ATQ.Height := 150;
ATQ.Length := 800; //1200;
ATQ.Weight := 1500;
ATQ.Width := 800;
ATQ.LabelPresent := 1;
ATQ.Label := CONCAT('TESTLABEL_',NewID);

fbITC_ManagerEmulation.M_AddData(
	meChannelSrc := 0,
	mMsgType     := E_ITC_MsgTypeConv.E_ADD_TU_REQUEST,
	mpData		 := ADR(ATQ),
    mLen 		 := SIZEOF(ATQ));

END_FUNCTION

// ---- 20_Product/20_ProBox/30_Toolbox/11_Emu/F_RemovePhysicalTU.TcPOU
FUNCTION F_RemovePhysicalTU : BOOL
(**************************************************************************************
 * 	Application		:	BoxControl Framework
 *	Revision		:	$Revision: 353897 $
 *	Revision date	:	$Date: 2015-08-24 22:28:50 +0200 (Mo, 24 Aug 2015) $
 *	Last changed by	:	$Author: d7mangc $
 *	URL				:	$URL: http://almscdc.swisslog.com/repo/SWPD/Development/BoxControlFramework/20_Release/trunk/01_Software/BoxControlFramework/BoxControlFramework/JumpStart/11_Library/10_Application/12_ElementFunctions/10_Functions/F_GetFunctionData.TcPOU $
 *
 *	Purpose			:	Removes physical (emulation) TU data
 *
 * ------------------------------------------------------------------------------------
 *	Copyright Swisslog [IP AG], Switzerland. All rights reserved.
 * 
 * ------------------------------------------------------------------------------------
 *	
 * 	Revision History: 
 *
 * 	VERSION			DATE			INITIALS			DESCRIPTION
 *	0.1				01.01.2001		swl					Example
 *
 **************************************************************************************)
VAR_INPUT
	eFunctionNumber : E_FunctionNumber;
	ZoneNumber		: INT;
END_VAR
VAR
	Name			: STRING;
	RTQ				: ST_ITC_RTQ;
	TransportData	: ST_TransportControlData;
END_VAR

TransportData := F_GetTransportControlData(eFunctionNumber, ZoneNumber);

IF TransportData.SensorOccupied THEN
	Name := F_GetFunctionName(eFunctionNumber:= eFunctionNumber, ZoneNumber:= ZoneNumber);
	RTQ.Position := F_ReduceToAlphaNumeric(InputString := Name);
	
	fbITC_ManagerEmulation.M_AddData(
		meChannelSrc := 0,
		mMsgType     := E_ITC_MsgTypeConv.E_REMOVE_TU_REQUEST,
		mpData		 := ADR(RTQ),
		mLen		 := SIZEOF(RTQ));
	
	F_RemovePhysicalTU := TRUE;
END_IF

END_FUNCTION

// ---- 20_Product/20_ProBox/30_Toolbox/70_Strategies/FB_CountTUs.TcPOU
FUNCTION_BLOCK FB_CountTUs
(**************************************************************************************
 * 	Application		:	BoxControl Framework
 *	Revision		:	$Revision: 411985 $
 *	Revision date	:	$Date: 2018-08-09 14:48:51 +0200 (Do., 09 Aug 2018) $
 *	Last changed by	:	$Author: p8fiscp $
 *	URL				:	$URL: http://almscdc.swisslog.com/repo/SWPD/Development/ProMove/02_Controls/ProBox/03_Implementation/01_DevelopmentProject/01_Software/ProBox_COE/ProBox_DevProj_v1.0/PLC_1/20_Product/10_App/12_E_Functions/11_ProBox/70_LoopControl/10_App/FB_ProBoxLoopCon $
 *
 *	Purpose			:	Count number of TU's inside the loop
 * ------------------------------------------------------------------------------------
 *	Copyright Swisslog [IP AG], Switzerland. All rights reserved.
 * 
 * ------------------------------------------------------------------------------------
 *	
 * 	Revision History: 
 *
 * 	VERSION			DATE			INITIALS			DESCRIPTION
 *	0.1				2018-06-01		PkF/RtK				First Version 
  *	0.2				2018-10-03		lca					Move NumberOfPallets to VAR_OUTPUT
 *
 **************************************************************************************)
VAR_INPUT
	Functions 				: ARRAY[1..E_FunctionNumber.F_END_FUNCTION] OF E_FunctionNumber;
	DestinationFunction		: E_FunctionNumber := E_FunctionNumber.F_BEGIN_FUNCTION;
	DestinationZone			: INT;
END_VAR

VAR_OUTPUT
	NumberOfTUs				: INT;
END_VAR

VAR
	Idx						: INT; 
	Idx2					: INT;
	NumberOfZones			: INT;	
	TransportControlData	: ST_TransportControlData;
	Destination				: ST_PositionIdent;
END_VAR


NumberOfTUs := 0;

FOR Idx := 1 TO E_FunctionNumber.F_END_FUNCTION DO
	IF Functions[Idx] <> E_FunctionNumber.F_END_FUNCTION THEN
		NumberOfZones := F_GetNumberOfZones(Functions[Idx]);
		FOR Idx2 := 1 TO NumberOfZones DO
			TransportControlData := F_GetTransportControlData(Functions[Idx],Idx2);
			// If the destination doesn't matter
			IF DestinationFunction = E_FunctionNumber.F_BEGIN_FUNCTION THEN
				NumberOfTUs := NumberOfTUs + UINT_TO_INT(TransportControlData.NumberOfPresentTUs);
			ELSE
				Destination := F_GetDestination(
						eFunctionNumber:= Functions[Idx] , 
						ZoneNumber:= Idx2, 
						DestinationIdx:= 1);
				// If the destination is correct		
				IF Destination.eFunctionNumber = DestinationFunction AND Destination.ZoneNumber = DestinationZone THEN
					NumberOfTUs := NumberOfTUs + UINT_TO_INT(TransportControlData.NumberOfPresentTUs);
				END_IF 
			END_IF
		END_FOR
	ELSE
		EXIT;
	END_IF
END_FOR

END_FUNCTION_BLOCK

// ---- 20_Product/20_ProBox/30_Toolbox/70_Strategies/FB_DTU_MergingControl.TcPOU
//DTU, transter unit Fifo control. Each side of the DTU is added to a fifo and DTU will choose the side as previous according to the FIFO
//if AutoTracking is enabled then check if the previus function has set the next functionnumber = DTU function number, it may be not ready, or the function is an output function from the DTU
FUNCTION_BLOCK FB_DTU_MergingControl //Driven Transfer Unit merging control
VAR_INPUT
		FunctionNumber 	: E_FunctionNumber;	// The function number of the transferUnit			
		DisableSide1	: BOOL;				// Optionally Disable adjacent side 1. if adjacent side is not used, then it is NOT mandatory to disable.  
		DisableSide2	: BOOL;				// Optionally Disable adjacent side 2. if adjacent side is not used, then it is NOT mandatory to disable.
		DisableSide3	: BOOL;				// Optionally Disable adjacent side 3. if adjacent side is not used, then it is NOT mandatory to disable.
		DisableSide4	: BOOL;				// Optionally Disable adjacent side 4. if adjacent side is not used, then it is NOT mandatory to disable.
		AutoTracking	: BOOL:=TRUE;		// Auto disables adjasent sides that do not set nextFunction to the DTU. Default enabled 
END_VAR

VAR_OUTPUT
	ePrevFunctionNumber	: E_FunctionNumber;	//the function number that has the highest priority to enter into Loop or intersection.	
END_VAR

VAR CONSTANT
	NUMBER_OF_ADJACENT_SIDES	: INT := 4;	
END_VAR

VAR	
	_fbFifo			:FB_MergingFiFo;	
	_Disabled		: ARRAY [1..NUMBER_OF_ADJACENT_SIDES] OF BOOL;			
	_ExternalFunction:E_FunctionNumber;
	_ExternalFuncSide:INT:=0;
END_VAR
VAR_TEMP
	i:INT;	
END_VAR


IF(FunctionNumber<=0 OR FunctionNumber>=E_FunctionNumber.F_BEGIN_EXTERN_FUNCTION) THEN RETURN; END_IF
IF( NOT __ISVALIDREF(FunctionRegistry[FunctionNumber].rSettingsFunction)) THEN RETURN; END_IF

//copy over user disable status to array.
_Disabled[1]:=DisableSide1;
_Disabled[2]:=DisableSide2;
_Disabled[3]:=DisableSide3;
_Disabled[4]:=DisableSide4;

 
//Run fifo control
FOR i:=1 TO NUMBER_OF_ADJACENT_SIDES BY 1 DO
	
	IF(AutoTracking) THEN
			_fbFifo.CompareNextFunc := FunctionNumber;
	ELSE
			_fbFifo.CompareNextFunc := E_FunctionNumber.F_BEGIN_FUNCTION; //Auto tracking is off
	END_IF
	_fbFifo(FunctionNumber:=FunctionRegistry[FunctionNumber].rSettingsFunction.eAdjacentFunctionNumberSide[i],Disable:=_Disabled[i]);	
END_FOR
//Run Fifo again to register external function (if supplied)
//CompareNextFunc argument should always be F_BEGIN_FUNCTION to disable tracking for external functions
IF(_ExternalFunction>E_FunctionNumber.F_BEGIN_FUNCTION AND _ExternalFuncSide>=0 AND _ExternalFuncSide<=NUMBER_OF_ADJACENT_SIDES) THEN	
	_fbFifo(FunctionNumber:=_ExternalFunction,Disable:=_Disabled[_ExternalFuncSide],CompareNextFunc:=E_FunctionNumber.F_BEGIN_FUNCTION);	
END_IF

//Set output
IF(_fbFifo.ePrevFunctionNumber = _ExternalFunction AND _ExternalFuncSide>0 AND _ExternalFuncSide < NUMBER_OF_ADJACENT_SIDES) THEN 
	ePrevFunctionNumber := FunctionRegistry[FunctionNumber].rSettingsFunction.eAdjacentFunctionNumberSide[_ExternalFuncSide];
ELSE
	ePrevFunctionNumber :=	_fbFifo.ePrevFunctionNumber;
END_IF

METHOD INTERNAL M_FindAdjacentSide : BOOL
VAR_INPUT
	AdjacentSide : E_FunctionNumber;
END_VAR
VAR_OUTPUT
	SideIndex:INT; // side 1,2,3 or 4
	ExternalFunction:BOOL; //The Function is a external Function assigned with M_SetExternalFunction
END_VAR
VAR
	i:INT;
END_VAR

//check that DTu_MergingControl is assigned to a DTU

IF(THIS^.FunctionNumber=0) THEN
	RETURN;
END_IF
IF(AdjacentSide=0) THEN
	RETURN;
END_IF

// Find the side on the DTU where the input function is oriented.
// check _ExternalFunction 
IF(_ExternalFunction = AdjacentSide) THEN
	SideIndex:= _ExternalFuncSide;
	ExternalFunction := TRUE;
	M_FindAdjacentSide:=TRUE;	
	RETURN;
END_IF

// Find the side on the DTU where the input function is oriented.
IF(__ISVALIDREF(FunctionRegistry[THIS^.FunctionNumber].rSettingsFunction)) THEN			
	FOR i:=1 TO NUMBER_OF_ADJACENT_SIDES BY 1 DO			
		//Get the DTU function number, where the input function is attached to
		IF( FunctionRegistry[THIS^.FunctionNumber].rSettingsFunction.eAdjacentFunctionNumberSide[i] = AdjacentSide)THEN
			SideIndex:= i;
			ExternalFunction := FALSE;
			M_FindAdjacentSide:=TRUE;
			EXIT;
		END_IF						 
	END_FOR
END_IF
END_METHOD

//Possible to set additional external function to a specific side
//This is used when DTU has an extended function on side 3-4
METHOD INTERNAL M_SetExternalFunction : BOOL
VAR_INPUT
	ExternalFunction	: E_FunctionNumber;
	ExternalFunctionSide:INT;
END_VAR
_ExternalFunction := ExternalFunction;
_ExternalFuncSide :=ExternalFunctionSide;
END_METHOD

END_FUNCTION_BLOCK

// ---- 20_Product/20_ProBox/30_Toolbox/70_Strategies/FB_LoopControl.TcPOU
FUNCTION_BLOCK PUBLIC FB_LoopControl
VAR_INPUT
	MaxTUsInLoop 			: INT:=30;
	AutoTracking			: BOOL:=TRUE;		//Default TRUE. Auto disables adjasent sides that do not set nextFunction to the DTU.
	InputTransferUnits		: ARRAY [0..GVL_STRATEGIES.MAX_TRANSFERUNITS] OF E_FunctionNumber;	//Array with all transfer units that has an input funciton connected
END_VAR
VAR_IN_OUT
	FunctionsInLoop			: ARRAY [*] OF E_FunctionNumber;	//Array with all functions in the loop (variable array length)
	InputFunctionsToLoop	: ARRAY [*] OF E_FunctionNumber;	//Array with all functions in the loop excluding InputTransferUnits (variable array length)	
END_VAR
VAR_OUTPUT
	TuCountInLoop 				: INT;
	LoopIsFull					: BOOL;
END_VAR
VAR CONSTANT		
	NUMBER_OF_ADJACENT_SIDES	: INT := 4;
END_VAR
VAR	
	_Init					: BOOL := FALSE;
	_InitRunning			: BOOL := FALSE;	
	_fbDTUMergingCtrl		: ARRAY [0..GVL_STRATEGIES.MAX_TRANSFERUNITS] OF FB_DTU_MergingControl;
	_Disables				: ARRAY [0..GVL_STRATEGIES.MAX_TRANSFERUNITS,1..NUMBER_OF_ADJACENT_SIDES] OF BOOL;
	_fbInFeedFunctionFifo	: FB_MergingFiFo;
	_StabilityCnt			: INT;
	_OverrideFunction		: E_FunctionNumber:=E_FunctionNumber.F_BEGIN_FUNCTION;
	//_ExternalFunction		: E_FunctionNumber:=E_FunctionNumber.F_BEGIN_FUNCTION; //possible additional external function to consider for an DTU
END_VAR

VAR_TEMP
	i:DINT;
	TUsInLoop				: INT;
	DTU_Disables			: ARRAY [0..GVL_STRATEGIES.MAX_TRANSFERUNITS,1..4] OF BOOL;
	DTU_NotReady			: BOOL;
	DTU_FunctionNumb		: E_FunctionNumber;
END_VAR

_M_Init();
//IF(NOT _Init) THEN RETURN; END_IF

//check if loop is full
TUsInLoop 		:=_M_CountTUsInLoop();
TuCountInLoop 	:= TUsInLoop;
LoopIsFull 		:= TUsInLoop >= MaxTUsInLoop;

//set prioirty (FIFO) for all input functions
FOR i:=LOWER_BOUND(InputFunctionsToLoop,1) TO UPPER_BOUND(InputFunctionsToLoop,1) BY 1 DO
	IF(InputFunctionsToLoop=0) THEN 
		EXIT; //pointer to array invalid, exit for loop
	ELSIF( InputFunctionsToLoop[i]<= E_FunctionNumber.F_BEGIN_FUNCTION OR InputFunctionsToLoop[i]>=E_FunctionNumber.F_END_FUNCTION) THEN
		EXIT; //no more functions to run
	ELSE
		DTU_NotReady := _M_CheckInfeedFunction(InputFunctionsToLoop[i],DTU_FuncNumb=>DTU_FunctionNumb);
		IF(AutoTracking) THEN
			_fbInFeedFunctionFifo.CompareNextFunc := DTU_FunctionNumb;
		ELSE
			_fbInFeedFunctionFifo.CompareNextFunc := E_FunctionNumber.F_BEGIN_FUNCTION; //Auto tracking is off
		END_IF
		_fbInFeedFunctionFifo(FunctionNumber:=InputFunctionsToLoop[i],Disable := DTU_NotReady);		
	END_IF
END_FOR

//If loop is full disable all input functions for DTU's
//If Loop is almost full, disable all but the most prioritized input function for DTU's
//Stability counter of 20 cycles added, just to be sure that if a transport from infeed function has started, it shall continue before choosing a new override function.
//TODO: Add dead lock protection, ie if the TU on OverrideFunction is not moved, then choose another input function. 
IF( TUsInLoop>= (MaxTUsInLoop-1)) THEN
	IF( TUsInLoop = (MaxTUsInLoop-1) AND _StabilityCnt >20) THEN	
		_OverrideFunction:=_fbInFeedFunctionFifo.ePrevFunctionNumber;
		_StabilityCnt:=0;
	ELSE
		_OverrideFunction:= F_BEGIN_FUNCTION;
	END_IF	
	_M_DisableInputFunctions(DTU_Disables:=DTU_Disables, OverrideInputFunction:=_OverrideFunction);
END_IF
IF(_StabilityCnt<=20) THEN
	_StabilityCnt:=_StabilityCnt+1;
END_IF

//Run each transfer unit Merging fifo control
FOR i:=0 TO GVL_STRATEGIES.MAX_TRANSFERUNITS BY 1 DO
	_fbDTUMergingCtrl[i](FunctionNumber:= InputTransferUnits[i],
						 DisableSide1:=_Disables[i,1] OR DTU_Disables[i,1],
						 DisableSide2:=_Disables[i,2] OR DTU_Disables[i,2],
						 DisableSide3:=_Disables[i,3] OR DTU_Disables[i,3],
						 DisableSide4:=_Disables[i,4] OR DTU_Disables[i,4],
						 AutoTracking:=AutoTracking	);
END_FOR

//Check DTU is ready,
//Return TRUE = Not Ready
//Return FALSE = Ready
METHOD PRIVATE _M_CheckInfeedFunction : BOOL
VAR_INPUT	
	InputFunctionToLoop  : E_FunctionNumber;
END_VAR
VAR_OUTPUT
	DTU_FuncNumb	: E_FunctionNumber;
END_VAR
VAR
	i				: INT;		
	Disable			: BOOL;	
	DTU_Ix			: INT;
	DTU_Side		: INT;
	ElementNumber	: E_ElementNumber;
	ExternalFunc	:BOOL; //The Function is a external Function assigned with M_SetExternalFunction
END_VAR

//CheckInfeedFunction

//Check if infeed function should be disabled
//Disable input function, ie set function to not available in FIFO
//Disabling input function if:
// -User has disabled the side on where the input function is located
// -DTU is occupied
// -DTU is in error.
// -DTU is disabled (by SIS telegram)
// 
DTU_FuncNumb:=0;

// Find the DTU and the side on the DTU where the input function is oriented.
FOR i:=0 TO GVL_STRATEGIES.MAX_TRANSFERUNITS BY 1 DO	
	IF(_fbDTUMergingCtrl[i].M_FindAdjacentSide(InputFunctionToLoop,SideIndex=>DTU_Side, ExternalFunction=>ExternalFunc)) THEN
		DTU_FuncNumb := _fbDTUMergingCtrl[i].FunctionNumber;
		DTU_Ix := i;				
		EXIT;
	END_IF	
END_FOR


//if DTU was found
IF(DTU_FuncNumb>E_FunctionNumber.F_BEGIN_FUNCTION AND DTU_Ix >= 0 AND DTU_Ix <= GVL_STRATEGIES.MAX_TRANSFERUNITS) THEN
	
	//Check if user has disabled the side on DTU where the infeed function is attached to
	Disable:=_Disables[DTU_Ix,DTU_Side];
	
	//Check if DTU already is occupied
	Disable:= Disable OR F_PB_GetTransportControlDataRef(DTU_FuncNumb,1).DataPresent;// OR F_PB_GetTransportControlDataRef(DTU,1).Occupied;
	
	//Check DTU has no active errors in element, functon or zones
	ElementNumber := FunctionRegistry[DTU_FuncNumb].rSettingsFunction.eElementLink;
	IF(__ISVALIDREF(ElementRegistry[ElementNumber].rElementData))THEN
		IF( ElementRegistry[ElementNumber].rElementData.ErrorData.FunctionErrorPending OR 
			ElementRegistry[ElementNumber].rElementData.ErrorData.ErrorState = E_ErrorState.ERROR) THEN
			Disable :=TRUE; //Error is present
		END_IF	
	END_IF	

	//Check if DTU is enabled
	Disable := Disable OR NOT F_CheckAllEnabled(DTU_FuncNumb);
END_IF

//Note, the MergingFifo control will check the infeed function if it self is operating, ie no error, enabled, ready to handover TU 

IF(ExternalFunc) THEN
	DTU_FuncNumb := E_FunctionNumber.F_BEGIN_FUNCTION;
END_IF
_M_CheckInfeedFunction:=Disable;
END_METHOD

METHOD PRIVATE _M_CountTUsInLoop : int
VAR_INPUT
END_VAR
VAR
	i:DINT;
	j:INT;
END_VAR

//count TU's for functions in "FunctionsInLoop" array
IF(FunctionsInLoop<>0) THEN	 //check pointer to array is valid 
	FOR i:=LOWER_BOUND(FunctionsInLoop,1) TO UPPER_BOUND(FunctionsInLoop,1) BY 1 DO	
		FOR j:=1 TO NUMBER_OF_ZONES_PER_FUNCTION BY 1 DO  //iterate through all zones		
			_M_CountTUsInLoop := _M_CountTUsInLoop + DINT_TO_INT(F_PB_GetTransportControlDataRef(FunctionsInLoop[i],j).NumberOfPresentTUs);		
		END_FOR
	END_FOR
END_IF

//count TU's for functions in "InputTransferUnits" array
FOR i:=0 TO  GVL_STRATEGIES.MAX_TRANSFERUNITS BY 1 DO			
	IF(InputTransferUnits[i] <> E_FunctionNumber.F_BEGIN_FUNCTION) THEN
		_M_CountTUsInLoop := _M_CountTUsInLoop + DINT_TO_INT(F_PB_GetTransportControlDataRef(InputTransferUnits[i],1(*onee zone only for DTUs*)).NumberOfPresentTUs);		
	END_IF
END_FOR 

//check that the inputTransferUnits are not in the FunctionsInLoop. ie mistake when entering functions in declaration of array variables 
IF(FunctionsInLoop<>0) THEN	//check pointer to array is valid
	FOR i:=LOWER_BOUND(FunctionsInLoop,1) TO UPPER_BOUND(FunctionsInLoop,1) BY 1 DO	
		FOR j:=0 TO GVL_STRATEGIES.MAX_TRANSFERUNITS BY 1 DO  //iterate through DTU's
			IF(FunctionsInLoop[i] =  InputTransferUnits[j]) THEN //yes, we have a bad configuration,(Input DTU also registered in functions in the loop) not a big deal, but we need to adjust the TU counter 		
				_M_CountTUsInLoop := _M_CountTUsInLoop - DINT_TO_INT(F_PB_GetTransportControlDataRef(InputTransferUnits[j],1(*onee zone only for DTUs*)).NumberOfPresentTUs);
			END_IF		
		END_FOR
	END_FOR
END_IF
END_METHOD

METHOD PRIVATE _M_DisableInputFunctions : BOOL
VAR_INPUT	
	OverrideInputFunction 	: E_FunctionNumber;
END_VAR
VAR_IN_OUT
	DTU_Disables			:ARRAY [0..GVL_STRATEGIES.MAX_TRANSFERUNITS,1..4] OF BOOL;
END_VAR
VAR
	i:INT;
	j:INT;
	k:DINT;
END_VAR

// Find the transfer unit where the inputfunctions belong to and disable the adjasent side
// If loop is almost full, it is possible to override the disable flag for an input function.

FOR i:=0 TO GVL_STRATEGIES.MAX_TRANSFERUNITS BY 1 DO	
	IF( InputTransferUnits[i]> 0 AND InputTransferUnits[i] < E_FunctionNumber.F_BEGIN_EXTERN_FUNCTION AND
		__ISVALIDREF(FunctionRegistry[InputTransferUnits[i]].rSettingsFunction)) THEN 
	
		FOR j:=1 TO NUMBER_OF_ADJACENT_SIDES BY 1 DO
			FOR k:=LOWER_BOUND(InputFunctionsToLoop,1) TO UPPER_BOUND(InputFunctionsToLoop,1) BY 1 DO
				IF(InputFunctionsToLoop=0) THEN EXIT; END_IF //pointer to array invalid, exit for loop
				IF(FunctionRegistry[InputTransferUnits[i]].rSettingsFunction.eAdjacentFunctionNumberSide[j] = InputFunctionsToLoop[k])THEN					
					DTU_Disables[i,j] := OverrideInputFunction <> InputFunctionsToLoop[k];
				END_IF
			END_FOR 
		END_FOR
	END_IF
	
END_FOR
END_METHOD

METHOD _M_Init : BOOL
VAR_INPUT
END_VAR
IF(NOT MainConv.Init) THEN
	_Init:=FALSE;	
	_InitRunning := FALSE;
END_IF

IF(NOT _Init AND _InitRunning) THEN
	_M_SanityCheck();	
	_init:=TRUE;
	_InitRunning := FALSE;
	
ELSIF(NOT _init) THEN
	_InitRunning:=TRUE;	
	//MainConv.fbDebugMsg.M_SendInfoMsg('Loop control init'); //Debug 	
END_IF
END_METHOD

(*
	Name: SanityCheck
	Description: 
		- Check that input functions are actually connected to a DTU
		- Check that all sides of a DTU is included in either loop functions or inputs to the loop functions
*)
METHOD PRIVATE _M_SanityCheck : BOOL
VAR
	i,j,k : DINT;
	InputDTUFound		: BOOL;				// An input DTU is found
	InputFuncFound		: BOOL;				// An input function is found
	LoopFuncFound		: BOOL;				// A loop function is found
	InputCheckValid		: BOOL := TRUE;	// Check at input has valid preliminary conditions
	InputDTUCheckValid	: BOOL := TRUE;	// Check at input DTU has valid preliminary conditions	
END_VAR


// Check that input functions are actually connected to a DTU
FOR i:=LOWER_BOUND(InputFunctionsToLoop,1) TO UPPER_BOUND(InputFunctionsToLoop,1) BY 1 DO
	IF(__ISVALIDREF(FunctionRegistry[InputFunctionsToLoop[i]].rSettingsFunction) AND __ISVALIDREF(FunctionRegistry[InputFunctionsToLoop[i]].rFunctionData)) THEN		
		InputDTUFound	:= FALSE;
		
		FOR j:=0 TO GVL_STRATEGIES.MAX_TRANSFERUNITS BY 1 DO
			InputDTUFound := _fbDTUMergingCtrl[j].M_FindAdjacentSide(InputFunctionsToLoop[i]);				
			// Match found, end further check at input function
			IF(InputDTUFound) THEN EXIT; END_IF
		END_FOR
				
		// Match not found for an input function, raise error
		IF(NOT InputDTUFound) THEN
			InputCheckValid := FALSE;
			F_SetError(
				ErrorType 	:= E_ErrorType.ERROR,
				ErrorParam 	:= 'Loop input not connected to Input DTU',
				ErrorMsg 	:= E_ErrorConv.CONFIGURATION_ERROR,
				ErrorData 	:= FunctionRegistry[InputFunctionsToLoop[i]].rFunctionData.ErrorData.ExternalError);
		END_IF
	END_IF
END_FOR


// Check that all sides of a DTU is included in either loop functions or inputs to the loop functions
FOR i:=0 TO GVL_STRATEGIES.MAX_TRANSFERUNITS BY 1 DO
	IF(__ISVALIDREF(FunctionRegistry[InputTransferUnits[i]].rSettingsFunction) AND __ISVALIDREF(FunctionRegistry[InputTransferUnits[i]].rFunctionData)) THEN
		InputFuncFound := FALSE;
		LoopFuncFound := FALSE;
		// Loop all adjacent sides
		FOR j:=1 TO 4 BY 1 DO
			// Find loop function on adjacent sides
			FOR k:=LOWER_BOUND(FunctionsInLoop,1) TO UPPER_BOUND(FunctionsInLoop,1) BY 1 DO
				IF(FunctionsInLoop[k] <> F_BEGIN_FUNCTION) THEN
					IF(FunctionRegistry[InputTransferUnits[i]].rSettingsFunction.eAdjacentFunctionNumberSide[j] = FunctionsInLoop[k]) THEN
						LoopFuncFound := TRUE;
						EXIT;
					END_IF
				END_IF
			END_FOR
			// Find Input function on adjacent sides
			FOR k:=LOWER_BOUND(InputFunctionsToLoop,1) TO UPPER_BOUND(InputFunctionsToLoop,1) BY 1 DO
				IF(InputFunctionsToLoop[k] <> F_BEGIN_FUNCTION) THEN
					IF(FunctionRegistry[InputTransferUnits[i]].rSettingsFunction.eAdjacentFunctionNumberSide[j] = InputFunctionsToLoop[k]) THEN
						InputFuncFound := TRUE;
						EXIT;
					END_IF
				END_IF
			END_FOR
		END_FOR
		// No matches found for a DTU, raise error
		IF(NOT(LoopFuncFound OR InputFuncFound)) THEN
			InputDTUCheckValid := FALSE;
			F_SetError(
				ErrorType 	:= E_ErrorType.ERROR,
				ErrorParam 	:= 'Input DTU not connected to loop or loop input',
				ErrorMsg 	:= E_ErrorConv.CONFIGURATION_ERROR,
				ErrorData 	:= FunctionRegistry[InputTransferUnits[i]].rFunctionData.ErrorData.ExternalError);
		// Only loop functions were not found, raise error
		ELSIF(NOT LoopFuncFound) THEN
			InputDTUCheckValid := FALSE;
			F_SetError(
				ErrorType 	:= E_ErrorType.ERROR,
				ErrorParam 	:= 'Input DTU not connected to loop',
				ErrorMsg 	:= E_ErrorConv.CONFIGURATION_ERROR,
				ErrorData 	:= FunctionRegistry[InputTransferUnits[i]].rFunctionData.ErrorData.ExternalError);
		// Only input functions were not found, raise error
		ELSIF(NOT InputFuncFound) THEN
			InputDTUCheckValid := FALSE;
			F_SetError(
				ErrorType 	:= E_ErrorType.ERROR,
				ErrorParam 	:= 'Input DTU not connected to loop input',
				ErrorMsg 	:= E_ErrorConv.CONFIGURATION_ERROR,
				ErrorData 	:= FunctionRegistry[InputTransferUnits[i]].rFunctionData.ErrorData.ExternalError);
		END_IF
	END_IF
END_FOR

_M_SanityCheck := InputCheckValid AND InputDTUCheckValid;
END_METHOD

METHOD PUBLIC M_DisableAdjasentSide
VAR_INPUT
	FunctionNumber 	: E_FunctionNumber;	// The transfer function number to witch the side is to be disabled.
	DisableSide1	: BOOL;				// Optionally Disable adjacent side 1. if adjacent side is not used, then it is NOT mandatory to disable.  
	DisableSide2	: BOOL;				// Optionally Disable adjacent side 2. if adjacent side is not used, then it is NOT mandatory to disable.
	DisableSide3	: BOOL;				// Optionally Disable adjacent side 3. if adjacent side is not used, then it is NOT mandatory to disable.
	DisableSide4	: BOOL;				// Optionally Disable adjacent side 4. if adjacent side is not used, then it is NOT mandatory to disable.
END_VAR
VAR
	i:INT;
END_VAR

FOR i:=0 TO GVL_STRATEGIES.MAX_TRANSFERUNITS BY 1 DO	
	
	IF(InputTransferUnits[i] = FunctionNumber) THEN
		_Disables[i,1] := DisableSide1;
		_Disables[i,2] := DisableSide2;
		_Disables[i,3] := DisableSide3;
		_Disables[i,4] := DisableSide4;
		EXIT;  //Quit
	END_IF
END_FOR
END_METHOD

METHOD PUBLIC M_GetPreviusFunction : E_FunctionNumber
VAR_INPUT
	FunctionNumber 	: E_FunctionNumber;	// The transfer function number to witch the prefered previus function shuld be returned.
END_VAR
VAR
	i:INT;
END_VAR

M_GetPreviusFunction:=E_FunctionNumber.F_BEGIN_FUNCTION;

FOR i:=0 TO GVL_STRATEGIES.MAX_TRANSFERUNITS BY 1 DO	
		IF(_fbDTUMergingCtrl[i].FunctionNumber = FunctionNumber) THEN
 			M_GetPreviusFunction :=_fbDTUMergingCtrl[i].ePrevFunctionNumber;
			EXIT;		
		END_IF
END_FOR
END_METHOD

//Add an additional function as a adjacent side
//Normally used for DTU's with extended function on axis 3.
//Only activeated during init
METHOD PUBLIC M_SetExternalFunction : BOOL
VAR_INPUT
	DtuFunctionNumber 	: E_FunctionNumber;	// The transfer function number to witch to set the external function.
	ExternalFunction	: E_FunctionNumber; // The External function to add as a "adjacent side"
	ExternalFunctionSide:INT; // The Side of the external function
END_VAR

VAR
	i:int;
END_VAR

IF(_init) THEN RETURN; END_IF

FOR i:=0 TO GVL_STRATEGIES.MAX_TRANSFERUNITS BY 1 DO		
	IF(_fbDTUMergingCtrl[i].FunctionNumber = DtuFunctionNumber) THEN
		_fbDTUMergingCtrl[i].M_SetExternalFunction(ExternalFunction,ExternalFunctionSide);		
		EXIT;  //Quit
	END_IF
END_FOR
END_METHOD

END_FUNCTION_BLOCK

// ---- 20_Product/20_ProBox/30_Toolbox/70_Strategies/F_PB_RoutingSlugging.TcPOU
(*
Standard routing on slugging functions.
Returns true if pallet(s) behind are headed towards this function and front is clear.
Returns false if pallet(s) behind are headed towards this function or front is not clear.
*)
FUNCTION F_PB_RoutingSlugging : BOOL
(**************************************************************************************
 * 	Application		:	BoxControl Framework
 *	Revision		:	$Revision: $
 *	Revision date	:	$Date: $
 *	Last changed by	:	$Author: $
 *	URL				:	$$
 *
 *	Purpose			:	Standard routing on slugging functions
 * ------------------------------------------------------------------------------------
 *	Copyright Swisslog [IP AG], Switzerland. All rights reserved.
 * 
 * ------------------------------------------------------------------------------------
 *	
 * 	Revision History: 
 *
 * 	VERSION			DATE			INITIALS			DESCRIPTION
 *	0.1				2018-11-15		PkF				First Version 
 *
 **************************************************************************************)
VAR_INPUT
		eFunctionNumber				: E_FunctionNumber; 				// Functions own function number
		RoutingSluggingData			: ST_RoutingSluggingData;
		OverrideTransport			: BOOL; 							// Override standard functionallity
		HoldTransport				: BOOL; 							// Hold transport
END_VAR

VAR
	LastZoneData					: ST_ZoneData;
	FirstZoneData					: ST_ZoneData;	
	OkTransport						: BOOL;
	NoPalletsBehind					: BOOL;
	NoPalletsInfront				: BOOL;
	Idx								: INT; // Loop var
	Idx2							: INT; // Loop var for Zones
	Idx3							: INT; // Loop var for invalid destinations check
	TransportControlData			: ST_TransportControlData;
	NumberOfZones					: INT;
	Destination						: E_FunctionNumber;
	TransportOK						: BOOL; // OK to run transport
END_VAR

// Get My Zone Data
LastZoneData 		:= F_GetZoneData(eFunctionNumber,F_GetNumberOfZones(eFunctionNumber));
FirstZoneData 		:= F_GetZoneData(eFunctionNumber,1);
// Init vars
OkTransport 		:= FALSE;
NoPalletsBehind 	:= TRUE;
NoPalletsInfront 	:= TRUE;

IF(HoldTransport) THEN
	RETURN;	// Return False
END_IF

IF ((LastZoneData.TransportControlData.Occupied) OR  OverrideTransport) THEN
	OKTransport	 := TRUE;	
	
ELSIF( FirstZoneData.TransportControlData.Occupied )THEN
	// Check behind
	FOR Idx := 1 TO 20 DO
		NumberOfZones := F_GetNumberOfZones(RoutingSluggingData.FunctionsBehind[Idx]);		
		// Note: NumberOfZones = 0 if FunctionsBehind[Idx] = E_FunctionNumber.F_BEGIN_FUNCTION		
		FOR Idx2 := 1 TO NumberOfZones DO
			TransportControlData := F_GetTransportControlData(RoutingSluggingData.FunctionsBehind[Idx],Idx2);

			IF 	TransportControlData.eTransportState = E_TransportState.TAKEOVER OR 
				TransportControlData.eTransportState = E_TransportState.FREE OR 
				TransportControlData.eTransportState = E_TransportState.IDLE OR 
				F_IsFunctionErrorPending(RoutingSluggingData.FunctionsBehind[Idx]) THEN
				;	// Function is considered empty	
			ELSE
				NoPalletsBehind := FALSE;	// Function is considered not empty (ie occupied) => wait for more pallets...
				// Check if destination of pallet is in the invalid list
				FOR Idx3 := 1 TO 20 DO
					Destination := F_PB_GetTuDestination(RoutingSluggingData.FunctionsBehind[Idx], Idx2, 1);
					
					IF 	Destination = RoutingSluggingData.InvalidDestinations[Idx3] AND
						Destination <> F_BEGIN_FUNCTION THEN
						NoPalletsBehind := TRUE;	// Function is considered empty
						EXIT;
					END_IF
				END_FOR
			END_IF
		END_FOR		
		
		//Exit for loop if desition already taken
		IF(NoPalletsBehind=FALSE) THEN
			EXIT; //exit for loop
		END_IF
	END_FOR
	
	// Check Forward
	FOR Idx := 1 TO 20 DO
		NumberOfZones := F_GetNumberOfZones(RoutingSluggingData.FunctionsInfront[Idx]);		
		// Note: NumberOfZones = 0 if FunctionsInfront[Idx] = E_FunctionNumber.F_BEGIN_FUNCTION
		FOR Idx2 := 1 TO NumberOfZones DO
			TransportControlData := F_GetTransportControlData(RoutingSluggingData.FunctionsInfront[Idx],Idx2);			
			IF TransportControlData.eTransportState = E_TransportState.TAKEOVER OR 
				TransportControlData.eTransportState = E_TransportState.FREE OR 
				TransportControlData.eTransportState = E_TransportState.IDLE THEN
				;	// Function is considered empty	
			ELSE
				NoPalletsInFront := FALSE;	// Function is considered not empty
			END_IF			
		END_FOR		
	END_FOR
	// OK to go, no pallets either behind or infront
	OkTransport := NoPalletsBehind AND NoPalletsInfront;
END_IF

F_PB_RoutingSlugging := OkTransport;

END_FUNCTION

// ---- 20_Product/20_ProBox/30_Toolbox/71_SafetyInterface/01_AK_Cabinet/FB_SafetySignalsAK.TcPOU
FUNCTION_BLOCK FB_SafetySignalsAK
VAR_INPUT
	SZPCo			: BOOL; //Safety Zone Pallet Conveyor 1	
	//NrOfContactor 	: INT :=3;//Number of contactors in cabinet
END_VAR
VAR_OUTPUT
END_VAR
VAR_IN_OUT
	SGref			: FB_ProBOXSG; //Reference to Switching group
	AKSignals		: ST_ProBoxSafetyAK;
END_VAR
VAR
	//fbBlink_1s	: FB_GeneratePulse := (Start := TRUE, PulseTimeOn := T#1S, PulseTimeOff := T#1S); // Blink 1s
	i,iMax		: INT;
	EmgStatus	: ST_EmgStatus;
END_VAR

//check if ResetSafetyNeeded
EmgStatus.eExternal := SZPCo;
EmgStatus.eInternal := AKSignals.Inputs.EsOk;
EmgStatus.eInternError := (AKSignals.Inputs.ComErr OR AKSignals.Inputs.FBErr); 
SGref.M_SetEmgStatus(EmgStatus);

//Pass signals from input to output
AKSignals.Outputs.ContactorOn 	:= SGref.CtrlOut.OpSummary.OpMcOn;
AKSignals.Outputs.ContactorOff 	:= SGref.CtrlOut.OpSummary.OpMcOff;
AKSignals.Outputs.ErrorAck 		:= SGref.CtrlOut.OpSummary.OpResetSafety;

// Copy over all feedback signals from SG group to be transfered to Safety							   
MEMCPY(ADR(AKSignals.Outputs.FeedBackContactor),ADR(SGref.HW_Inputs.Diag.FeedbackMainContactorOFF),SIZEOF(AKSignals.Outputs.FeedBackContactor));

END_FUNCTION_BLOCK

// ---- 20_Product/20_ProBox/30_Toolbox/71_SafetyInterface/02_LowLift/FB_SafetySignalsLowLift.TcPOU
FUNCTION_BLOCK FB_SafetySignalsLowLift
VAR_INPUT
	SZPCo			:BOOL; //Safety Zone Pallet Conveyor 1
END_VAR
VAR_OUTPUT
END_VAR
VAR_IN_OUT
	LowLiftSignals	:	ST_ProBoxSafetyLowLift;
END_VAR
VAR
	fbBlink_1s	: FB_GeneratePulse := (Start := TRUE, PulseTimeOn := T#1S, PulseTimeOff := T#1S); // Blink 1s
	i			: INT;
END_VAR

fbBlink_1s();

//Indicate that an error exit with blinking blue lamp on cabinet. 
IF fbBlink_1s.Pulse AND (LowLiftSignals.Inputs.ComErr OR LowLiftSignals.Inputs.FBErr) OR NOT LowLiftSignals.Inputs.EsOk OR NOT LowLiftSignals.Inputs.LightGridOk THEN
	LowLiftSignals.Outputs.ResetSafetyNeeded := TRUE;
ELSE 
	LowLiftSignals.Outputs.ResetSafetyNeeded := FALSE;
END_IF

//Indicate that lowlift have been reseted but main contactors not pulled
IF NOT LowLiftSignals.Outputs.ResetSafetyNeeded AND  LowLiftSignals.Inputs.FeedBackK1 AND LowLiftSignals.Inputs.FeedBackK2 THEN
	LowLiftSignals.Outputs.ResetSafetyNeeded := fbBlink_1s.Pulse;	
END_IF
//Pass signals from input to output
LowLiftSignals.Outputs.ContactorOn := LowLiftSignals.Inputs.ContactorOn;
LowLiftSignals.Outputs.ContactorOff := LowLiftSignals.Inputs.ContactorOff;
LowLiftSignals.Outputs.FeedBackK1 := LowLiftSignals.Inputs.FeedBackK1;
LowLiftSignals.Outputs.FeedBackK2 := LowLiftSignals.Inputs.FeedBackK2;

//Pass on pushbutton and pass on to Safety
LowLiftSignals.Outputs.ErrorAck := LowLiftSignals.Inputs.ResetSafety;

END_FUNCTION_BLOCK

// ---- 20_Product/20_ProBox/30_Toolbox/71_SafetyInterface/03_Shuttle/FB_SafetySignalsShuttle.TcPOU
FUNCTION_BLOCK FB_SafetySignalsShuttle
VAR_INPUT
	SZPCo				: BOOL; //Safety Zone Pallet Conveyor 1	
	AP_Shuttle_Index	: INT :=1; //Index in SG AP array that is used for the cabinet on the shuttle car 	
END_VAR
VAR_OUTPUT
END_VAR
VAR_IN_OUT
	SGref			:  	FB_ProBOXSG; //Inputs from Switching group
	ShuttleSignals	:	ST_ProBoxSafetyShuttle;
END_VAR
VAR	
	EmgStatus		: ST_EmgStatus;
END_VAR

//check if ResetSafetyNeeded
EmgStatus.eExternal := SZPCo;
EmgStatus.eInternal := ShuttleSignals.Inputs.EsOk;
EmgStatus.eInternError := (ShuttleSignals.Inputs.ComErr OR ShuttleSignals.Inputs.FBErr); 
SGref.M_SetEmgStatus(EmgStatus);


//Pass signals from input to output
IF(AP_Shuttle_Index >0 AND AP_Shuttle_Index<= GVL_PB_SG.NUMBER_OF_CONTACTORS) THEN
	ShuttleSignals.Outputs.ContactorOnShuttle := SGref.HW_Inputs.AP[AP_Shuttle_Index].OpMcOn;  //get the specific contactor ON button on the shuttle cabinet
END_IF
ShuttleSignals.Outputs.ContactorOnEntry := SGref.CtrlOut.OpSummary.OpMcOn;
ShuttleSignals.Outputs.EmergencyDrive 	:= SGref.CtrlOut.OpSummary.OpEmgDrive;
ShuttleSignals.Outputs.ErrorAck 		:= SGref.CtrlOut.OpSummary.OpResetSafety;


// Copy over all feedback signals from SG group to be transfered to Safety							   
MEMCPY(ADR(ShuttleSignals.Outputs.FeedBackContactor),ADR(SGref.HW_Inputs.Diag.FeedbackMainContactorOFF),SIZEOF(ShuttleSignals.Outputs.FeedBackContactor));

END_FUNCTION_BLOCK

// ---- 20_Product/20_ProBox/30_Toolbox/71_SafetyInterface/04_VerticalConveyor/FB_SafetySignalsVerticalConv.TcPOU
FUNCTION_BLOCK FB_SafetySignalsVerticalConv
VAR_INPUT
	SZPCo						: BOOL; //Safety Zone Pallet Conveyor	
END_VAR
VAR_IN_OUT
	SGref			: FB_ProBOXSG; //Reference to Switching group
	VCSignals		: ST_ProBoxSafetyVerticalConv;
END_VAR
VAR
	EmgStatus		: ST_EmgStatus;
END_VAR

//check if ResetSafetyNeeded
EmgStatus.eExternal := SZPCo;
EmgStatus.eInternal := VCSignals.Inputs.EsOk AND VCSignals.Inputs.VcOK;
EmgStatus.eInternError := (VCSignals.Inputs.ComErr OR VCSignals.Inputs.FBErr); 
SGref.M_SetEmgStatus(EmgStatus);


//Pass signals from input to output
VCSignals.Outputs.ContactorOn 		:= SGref.CtrlOut.OpSummary.OpMcOn;
VCSignals.Outputs.ContactorOff 		:= SGref.CtrlOut.OpSummary.OpMcOff;
VCSignals.Outputs.ErrorAck 			:= SGref.CtrlOut.OpSummary.OpResetSafety;
                                                              
VCSignals.Outputs.EmergencyDrive	:= SGref.CtrlOut.OpSummary.OpEmgDrive;
VCSignals.Outputs.ManAuto 			:= SGref.CtrlOut.OpSummary.OpManAuto;
VCSignals.Outputs.EntryRequest 		:= SGref.CtrlOut.OpSummary.OpEntryReq;
//VerticalConvSignals.Outputs.DoorClosed := HW_ElementSignalsToGroup.DoorClosed;


// Copy over all feedback signals from SG group to be transfered to Safety							   
MEMCPY(ADR(VCSignals.Outputs.FeedBackContactor),ADR(SGref.HW_Inputs.Diag.FeedbackMainContactorOFF),SIZEOF(VCSignals.Outputs.FeedBackContactor));

END_FUNCTION_BLOCK

// ---- 20_Product/20_ProBox/30_Toolbox/71_SafetyInterface/SafetyZoneSignals/FB_SafetySignalsSZPCo.TcPOU
FUNCTION_BLOCK FB_SafetySignalsSZPCo
VAR_INPUT
	ErrorAck		: BOOL; //Summarized from all reset safety buttons located within safety zone
END_VAR
VAR_OUTPUT
	TwinSafeError	: BOOL; //Error in FB or Com in TwinSafe
	TwinSafeOK		: BOOL; //Summary of Safety zone inputs
END_VAR
VAR_IN_OUT
	SZPCoSignals	:	ST_ProBoxSafetySZPCo;
END_VAR
VAR	
	i			: INT;
END_VAR

//Indicate that an error exit with blinking blue lamp on cabinet. 
IF (SZPCoSignals.Inputs.ComErr OR SZPCoSignals.Inputs.FBErr) THEN
	TwinSafeError := TRUE;
ELSE 
	TwinSafeError := FALSE;
END_IF

TwinSafeOK := SZPCoSignals.Inputs.SafetyZoneOk AND NOT TwinSafeError;

//Pass on pushbutton and pass on to Safety
SZPCoSignals.Outputs.ErrorAck := ErrorAck;

END_FUNCTION_BLOCK

// ---- 20_Product/20_ProBox/30_Toolbox/FB_ClockHz.TcPOU
PROGRAM FB_ClockHz
(**************************************************************************************
 *  Application     :   ProBoxControl Framework
 *  Revision        :   $Revision: 334272 $
 *  Revision date   :   $Date: 2013-09-23 11:26:06 +0200 (Wed, 23 Sep 2015) $
 *  Last changed by :   $Author: b7test $
 *  URL             :   $URL: $
 * ------------------------------------------------------------------------------------
 *  © Swisslog AG
 *  Swisslog is not liable for any usage of this source code that is not agreed 
 *  on between Swisslog and the other party. The mandatory legal liability remains 
 *  unaffected.
 * ------------------------------------------------------------------------------------
 *  Revision History: 
 *
 *  VERSION         DATE            INITIALS            DESCRIPTION
 *  0.1             14.11.2018      RnK                 Clock Pulse
 *
 **************************************************************************************)

VAR
	{attribute 'hide'}	fb05Hz			: TON; //Timer for positive flank
	{attribute 'hide'}	fb05HzInv		: TON; //Timer for negative flank
	
	{attribute 'hide'}	n1HzCounter		: UINT; //Counter for 1Hz internal use
	{attribute 'hide'}	n2HzCounter		: UINT; //Counter for 2Hz internal use
	{attribute 'hide'}	n5HzCounter		: UINT; //Counter for 5Hz internal use
	{attribute 'hide'}	n10HzCounter	: UINT; //Counter for 10Hz internal use
END_VAR
	
VAR_OUTPUT	
	Clock_1Hz			: BOOL;	// 1s pulse
	Clock_2Hz			: BOOL;	// 2s pulse
	Clock_5Hz			: BOOL;	// 5s pulse
	Clock_10Hz			: BOOL;	// 10s pulse
END_VAR

// Timer for 500ms Hz
	fb05Hz(IN:= NOT fb05HzInv.Q, PT:= T#50MS, Q=> Clock_10Hz);
	fb05HzInv(IN:= fb05Hz.Q, PT:= T#50MS);

// Counter used for different Hz	
	IF 	Clock_10Hz AND fb05HzInv.Q THEN // Will add 1 to a counter each 500ms on positive flank
		n5HzCounter := n5HzCounter + 1;
		n2HzCounter := n2HzCounter + 1;
		n1HzCounter := n1HzCounter + 1;
		n10HzCounter := n10HzCounter + 1;
	END_IF
	
// 1Hz Clock Pulse
	IF	n5HzCounter < 1 THEN
		Clock_5Hz := TRUE;
	ELSIF
		n1HzCounter < 2 THEN
		Clock_5Hz := FALSE;
	ELSE 
		n5HzCounter := 0;
	END_IF

	
// 2Hz Clock Pulse
	IF	n2HzCounter < 2 THEN
		Clock_2Hz := TRUE;
	ELSIF
		n2HzCounter < 4 THEN
		Clock_2Hz := FALSE;
	ELSE 
		n2HzCounter := 0;
	END_IF

	
// 5Hz Clock Pulse
	IF	n1HzCounter < 5 THEN
		Clock_1Hz := TRUE;
	ELSIF
		n1HzCounter >= 5 THEN
		Clock_1Hz := FALSE;
		END_IF
	IF n1HzCounter >= 10 THEN
		n1HzCounter :=0;
	END_IF

END_PROGRAM

// ---- 20_Product/20_ProBox/30_Toolbox/FB_CountTUDestination.TcPOU
FUNCTION_BLOCK FB_CountTUDestination
(**************************************************************************************
 * 	Application		:	BoxControl Framework
 *	Revision		:	$Revision: 411985 $
 *	Revision date	:	$Date: 2018-08-09 14:48:51 +0200 (Do., 09 Aug 2018) $
 *	Last changed by	:	$Author: q8ottoc $
 *	URL				:	$URL: http://almscdc.swisslog.com/repo/SWPD/Development/ProMove/02_Controls/ProBox/03_Implementation/01_DevelopmentProject/01_Software/ProBox_COE/ProBox_DevProj_v1.0/PLC_1/20_Product/10_App/12_E_Functions/11_ProBox/70_LoopControl/10_App/FB_ProBoxLoopCon $
 *
 *	Purpose			:	Count number of TU's destination inside loop
 * ------------------------------------------------------------------------------------
 *	Copyright Swisslog [IP AG], Switzerland. All rights reserved.
 * 
 * ------------------------------------------------------------------------------------
 *	
 * 	Revision History: 
 *
 * 	VERSION			DATE			INITIALS			DESCRIPTION
 *	0.1				2018-06-01		PkF/RtK				First Version 
  *	0.2				2018-10-03		lca					Move NumberOfPallets to VAR_OUTPUT
 *
 **************************************************************************************)
VAR_INPUT
	Functions 				: ARRAY[1..E_FunctionNumber.F_END_FUNCTION] OF E_FunctionNumber;
	DestinationFunction1	: E_FunctionNumber := E_FunctionNumber.F_10_001_1122_01_0;
	DestinationFunction2	: E_FunctionNumber := E_FunctionNumber.F_10_002_1061_01_0;
	DestinationFunction3	: E_FunctionNumber := E_FunctionNumber.F_10_002_1065_01_0;	
	DestinationZone			: INT;
END_VAR

VAR_OUTPUT
	NumberOfTUsDest1		: INT;
	NumberOfTUsDest2		: INT;
	NumberOfTUsDest3		: INT;	
END_VAR

VAR
	Idx						: INT; 
	Idx2					: INT;
	NumberOfZones			: INT;	
	TransportControlData	: ST_TransportControlData;
	Destination				: ST_PositionIdent;
END_VAR


NumberOfTUsDest1 := 0;
NumberOfTUsDest2 := 0;
NumberOfTUsDest3 := 0;

FOR Idx := 1 TO E_FunctionNumber.F_END_FUNCTION DO
	IF Functions[Idx] <> E_FunctionNumber.F_END_FUNCTION THEN
		NumberOfZones := F_GetNumberOfZones(Functions[Idx]);
		FOR Idx2 := 1 TO NumberOfZones DO
			TransportControlData := F_GetTransportControlData(Functions[Idx],Idx2);
			// If the destination doesn't matter
			Destination := F_GetDestination(
						eFunctionNumber:= Functions[Idx] , 
						ZoneNumber:= Idx2, 
						DestinationIdx:= 1);
				// If the destination is correct		
				IF Destination.eFunctionNumber = DestinationFunction1 THEN
					NumberOfTUsDest1 := NumberOfTUsDest1 + UINT_TO_INT(TransportControlData.NumberOfPresentTUs);
				END_IF 
				IF Destination.eFunctionNumber = DestinationFunction2 THEN
					NumberOfTUsDest2 := NumberOfTUsDest2 + UINT_TO_INT(TransportControlData.NumberOfPresentTUs);
				END_IF 
				IF Destination.eFunctionNumber = DestinationFunction3 THEN
					NumberOfTUsDest3 := NumberOfTUsDest3 + UINT_TO_INT(TransportControlData.NumberOfPresentTUs);
				END_IF 
		END_FOR
	END_IF
END_FOR

END_FUNCTION_BLOCK

// ---- 20_Product/20_ProBox/30_Toolbox/FB_FunctionOrdersToProBox.TcPOU
FUNCTION_BLOCK FB_FunctionOrdersToProBox
VAR_INPUT
	FunctionOrders : ST_FunctionOrders;
END_VAR

VAR_OUTPUT
	Speed_12 		: E_ProBoxMotorSpeed;
	Direction_12	: E_ProBoxMotorDirection;
	Run_12			: BOOL;
	Enable_12		: BOOL;
	Speed_34 		: E_ProBoxMotorSpeed;
	Direction_34	: E_ProBoxMotorDirection;
	Run_34			: BOOL;
	Enable_34		: BOOL;	
END_VAR

VAR
END_VAR

IF FunctionOrders.ReqSpeed > 50 THEN
	Speed_12 := E_ProBoxMotorSpeed.NORMAL;
ELSIF FunctionOrders.ReqSpeed > 20 AND FunctionOrders.ReqSpeed <= 50 THEN
	Speed_12 := E_ProBoxMotorSpeed.LOW_SPEED;
ELSE
	Speed_12 := E_ProBoxMotorSpeed.CREEP_SPEED;
END_IF

IF FunctionOrders.ReqSpeed_34 > 50 THEN
	Speed_34 := E_ProBoxMotorSpeed.NORMAL;
ELSIF FunctionOrders.ReqSpeed_34 > 20 AND FunctionOrders.ReqSpeed_34 <= 50 THEN
	Speed_34 := E_ProBoxMotorSpeed.LOW_SPEED;
ELSE
	Speed_34 := E_ProBoxMotorSpeed.CREEP_SPEED;
END_IF

IF FunctionOrders.ReqDriveDirection THEN
	Direction_12 := E_ProBoxMotorDirection.MOTOR_FORWARD;
ELSE
	Direction_12 := E_ProBoxMotorDirection.MOTOR_REVERSE;
END_IF

IF FunctionOrders.ReqDriveDirection_34 THEN
	Direction_34 := E_ProBoxMotorDirection.MOTOR_FORWARD;
ELSE
	Direction_34 := E_ProBoxMotorDirection.MOTOR_REVERSE;
END_IF

Run_12 := FunctionOrders.ReqDriveRun;
Run_34 := FunctionOrders.ReqDriveRun_34;

Enable_12 := FunctionOrders.Enable;
Enable_34 := FunctionOrders.Enable_34;

END_FUNCTION_BLOCK

// ---- 20_Product/20_ProBox/30_Toolbox/FB_PAC_CapacityCounter.TcPOU
FUNCTION_BLOCK FB_PAC_CapacityCounter
VAR_INPUT
	sNetId                : T_AmsNetId ;    (* TwinCAT system network address *)
    sFileName            : T_MaxString ;(* CSV destination file path and name *)
	EnableTime				: TIME;
	StartPACCounter			: BOOL:=FALSE;
	
	LogData01:E_FunctionNumber;
	LogData02:E_FunctionNumber;
	LogData03:E_FunctionNumber;
	LogData04:E_FunctionNumber;
	LogData05:E_FunctionNumber;
	LogData06:E_FunctionNumber;
	LogData07:E_FunctionNumber;
	LogData08:E_FunctionNumber;
	LogData09:E_FunctionNumber;
	LogData10:E_FunctionNumber;
	LogData11:E_FunctionNumber;
	LogData12:E_FunctionNumber;
	LogData13:E_FunctionNumber;
	LogData14:E_FunctionNumber;
	LogData15:E_FunctionNumber;
	LogData16:E_FunctionNumber;
	LogData17:E_FunctionNumber;
	LogData18:E_FunctionNumber;
	LogData19:E_FunctionNumber;
	LogData20:E_FunctionNumber;
END_VAR
VAR_OUTPUT
	Output: ARRAY [1..100] OF STRING;
	ActualTimerValue: Time;
END_VAR
VAR
	ResetPACCounter	: BOOL :=FALSE;
	LogData: ARRAY [1..100] OF INT;
	TransportCtrlData		: ARRAY[1..F_END_FUNCTION-1] OF ST_TransportControlData;
    sCSVLine            : ARRAY [1..1000000] OF BYTE;(* Single CSV text line (row, record), we are using string as record buffer (your are able to see created fields) *)
    sCSVField            : T_MaxString := '';(* Single CSV field value (column, record field) *)
    sTest                : T_MaxString :='Test';
    bBusy                : BOOL;
    bError                : BOOL;
    nErrId                : UDINT;
    nRow                 : UDINT     := 0;(* Row number (record) *)
    nColumn                : UDINT     := 0;(* Column number (record field) *)
   // hFile                : UINT        := 0;(* File handle of the source file *)
    step                : DWORD     := 0;
    fbFileOpen            : FB_FileOpen;(* Opens file *)
	fbFileSeek				: FB_FileSeek;
	fbFileRead			  : FB_FileRead;	
    fbFileClose            : FB_FileClose;(* Closes file *)
    fbFileWrite            : FB_FileWrite;(* Writes one record (line) *)
    fbWriter            : FB_CSVMemBufferWriter;(* Helper function block used to create CSV data bytes (single record line) *)
    str_Output: STRING;
    fbFormat        : FB_FormatString;
 
	tTimeOut                        : TIME := DEFAULT_ADS_TIMEOUT;
	TotalTime: STRING;
	
	CounterPosition01: CTU;
	CounterPosition02: CTU;
	CounterPosition03: CTU;
	CounterPosition04: CTU;
	CounterPosition05: CTU;
	CounterPosition06: CTU;
	CounterPosition07: CTU;
	CounterPosition08: CTU;
	CounterPosition09: CTU;
	CounterPosition10: CTU;
	CounterPosition11: CTU;
	CounterPosition12: CTU;
	CounterPosition13: CTU;
	CounterPosition14: CTU;
	CounterPosition15: CTU;
	CounterPosition16: CTU;
	CounterPosition17: CTU;
	CounterPosition18: CTU;
	CounterPosition19: CTU;
	CounterPosition20: CTU;
	
	Ton1:TON;
	Ton2:TON;

	FileReady : BOOL;

	EnableT: BOOL;
	bReadReady: BOOL;
	SourcehFile: UINT := 0;
	DestinationhFile: UINT := 0;
	Wait : TOF;
	fbLocalTime: FB_LocalSystemTime;
	GetLocalTime : BOOL;
	sSystemTime : TIMESTRUCT;

END_VAR

TransportCtrlData[LogData01]:= F_GetTransportControlData(LogData01,1);
TransportCtrlData[LogData02]:= F_GetTransportControlData(LogData02,1);
TransportCtrlData[LogData03]:= F_GetTransportControlData(LogData03,1);
TransportCtrlData[LogData04]:= F_GetTransportControlData(LogData04,1);
TransportCtrlData[LogData05]:= F_GetTransportControlData(LogData05,1);
TransportCtrlData[LogData06]:= F_GetTransportControlData(LogData06,1);
TransportCtrlData[LogData07]:= F_GetTransportControlData(LogData07,1);
TransportCtrlData[LogData08]:= F_GetTransportControlData(LogData08,1);
TransportCtrlData[LogData09]:= F_GetTransportControlData(LogData09,1);
TransportCtrlData[LogData10]:= F_GetTransportControlData(LogData10,1);
TransportCtrlData[LogData11]:= F_GetTransportControlData(LogData11,1);
TransportCtrlData[LogData12]:= F_GetTransportControlData(LogData12,1);
TransportCtrlData[LogData13]:= F_GetTransportControlData(LogData13,1);
TransportCtrlData[LogData14]:= F_GetTransportControlData(LogData14,1);
TransportCtrlData[LogData15]:= F_GetTransportControlData(LogData15,1);
TransportCtrlData[LogData16]:= F_GetTransportControlData(LogData16,1);
TransportCtrlData[LogData17]:= F_GetTransportControlData(LogData17,1);
TransportCtrlData[LogData18]:= F_GetTransportControlData(LogData18,1);
TransportCtrlData[LogData19]:= F_GetTransportControlData(LogData19,1);
TransportCtrlData[LogData20]:= F_GetTransportControlData(LogData20,1);

fbLocalTime(
	sNetID:= sNetId, 
	bEnable:= TRUE, 
	dwCycle:= 1 , 
	dwOpt:= , 
	tTimeout:= , 
	bValid=> GetLocalTime, 
	systemTime=>sSystemTime , 
	tzID=> );


// Timer For Counter
Ton1(IN:=StartPACCounter AND NOT (Ton1.ET=Ton1.PT),PT:=EnableTime); // *************************change the timer according to requirement ******************************
(*IF StartPACCounter THEN
	EnableT:=TRUE;
END_IF*)
ActualTimerValue:=Ton1.ET;
TotalTime:=SYSTEMTIME_TO_STRING(fbLocalTime.systemTime);

// Log Data From Position one
CounterPosition01(CU:=TransportCtrlData[LogData01].Occupied,PV:=10000);
Output[1]:= 'TotalTime';
Output[2]:= TotalTime;//RIGHT(TOD_TO_STRING(TotalTime), 8);
Output[3]:= F_GetFunctionName(LogData01,1);
Output[4]:= WORD_TO_STRING(CounterPosition01.CV );

// Log Data From Position two
CounterPosition02(CU:=TransportCtrlData[LogData02].Occupied,PV:=10000);		
Output[5]:=F_GetFunctionName(LogData02,1);
Output[6]:=WORD_TO_STRING(CounterPosition02.CV);	
// Log Data From Position three
CounterPosition03(CU:=TransportCtrlData[LogData03].Occupied,PV:=10000);		
Output[7]:=F_GetFunctionName(LogData03,1);
Output[8]:=WORD_TO_STRING(CounterPosition03.CV);

// Log Data From Position Four
CounterPosition04(CU:=TransportCtrlData[LogData04].Occupied,PV:=10000);
Output[9]:=F_GetFunctionName(LogData04,1);
Output[10]:=WORD_TO_STRING(CounterPosition04.CV );

// Log Data From Position Five
CounterPosition05(CU:=TransportCtrlData[LogData05].Occupied,PV:=10000);		
Output[11]:=F_GetFunctionName(LogData05,1);
Output[12]:=WORD_TO_STRING(CounterPosition05.CV);
	
// Log Data From Position Six
CounterPosition06(CU:=TransportCtrlData[LogData06].Occupied,PV:=10000);		
Output[13]:=F_GetFunctionName(LogData06,1);
Output[14]:=WORD_TO_STRING(CounterPosition06.CV);

// Log Data From Position Seven
CounterPosition07(CU:=TransportCtrlData[LogData07].Occupied,PV:=10000);		
Output[15]:=F_GetFunctionName(LogData07,1);
Output[16]:=WORD_TO_STRING(CounterPosition07.CV);

// Log Data From Position Eight
CounterPosition08(CU:=TransportCtrlData[LogData08].Occupied,PV:=10000);
Output[17]:=F_GetFunctionName(LogData08,1);
Output[18]:=WORD_TO_STRING(CounterPosition08.CV );

// Log Data From Position Nine
CounterPosition09(CU:=TransportCtrlData[LogData09].Occupied,PV:=10000);		
Output[19]:=F_GetFunctionName(LogData09,1);
Output[20]:=WORD_TO_STRING(CounterPosition09.CV);
	
// Log Data From Position Ten
CounterPosition10(CU:=TransportCtrlData[LogData10].Occupied,PV:=10000);		
Output[21]:=F_GetFunctionName(LogData10,1);
Output[22]:=WORD_TO_STRING(CounterPosition10.CV);

// Log Data From Position one
CounterPosition11(CU:=TransportCtrlData[LogData11].Occupied,PV:=10000);
Output[23]:=  F_GetFunctionName(LogData11,1);
Output[24]:= WORD_TO_STRING(CounterPosition11.CV );

// Log Data From Position two
CounterPosition12(CU:=TransportCtrlData[LogData12].Occupied,PV:=10000);		
Output[25]:=F_GetFunctionName(LogData12,1);
Output[26]:=WORD_TO_STRING(CounterPosition12.CV);	

// Log Data From Position three
CounterPosition13(CU:=TransportCtrlData[LogData13].Occupied,PV:=10000);		
Output[27]:=F_GetFunctionName(LogData13,1);
Output[28]:=WORD_TO_STRING(CounterPosition13.CV);

// Log Data From Position Four
CounterPosition14(CU:=TransportCtrlData[LogData14].Occupied,PV:=10000);
Output[29]:=F_GetFunctionName(LogData14,1);
Output[30]:=WORD_TO_STRING(CounterPosition14.CV );

// Log Data From Position Five
CounterPosition15(CU:=TransportCtrlData[LogData15].Occupied,PV:=10000);		
Output[31]:=F_GetFunctionName(LogData15,1);
Output[32]:=WORD_TO_STRING(CounterPosition15.CV);
	
// Log Data From Position Six
CounterPosition16(CU:=TransportCtrlData[LogData16].Occupied,PV:=10000);		
Output[33]:=F_GetFunctionName(LogData16,1);
Output[34]:=WORD_TO_STRING(CounterPosition16.CV);

// Log Data From Position Seven
CounterPosition17(CU:=TransportCtrlData[LogData17].Occupied,PV:=10000);		
Output[35]:=F_GetFunctionName(LogData17,1);
Output[36]:=WORD_TO_STRING(CounterPosition17.CV);

// Log Data From Position Eight
CounterPosition18(CU:=TransportCtrlData[LogData18].Occupied,PV:=10000);
Output[37]:=F_GetFunctionName(LogData18,1);
Output[38]:=WORD_TO_STRING(CounterPosition18.CV );

// Log Data From Position Nine
CounterPosition19(CU:=TransportCtrlData[LogData19].Occupied,PV:=10000);		
Output[39]:=F_GetFunctionName(LogData19,1);
Output[40]:=WORD_TO_STRING(CounterPosition19.CV);
	
// Log Data From Position Ten
CounterPosition20(CU:=TransportCtrlData[LogData20].Occupied,PV:=10000);		
Output[41]:=F_GetFunctionName(LogData20,1);
Output[42]:=WORD_TO_STRING(CounterPosition20.CV);

CASE step OF
    0:    (* Wait for rising edge at bWrite variable *)
        IF Ton1.Q THEN
          //  bWrite         := FALSE;
            bBusy         := TRUE;
            bError        := FALSE;
            nErrId        := 0;
            SourcehFile        := 0;
			DestinationhFile        := 0;
            nRow         := 0;
            nColumn    := 0;
            step         := 1;
        END_IF
		
	1:    (*Open Source file*)
        fbFileOpen(  bExecute := FALSE  );
        fbFileOpen( sNetId := sNetId, sPathName := sFileName, nMode := FOPEN_MODEAPPEND OR FOPEN_MODEBINARY ,(* Open file in BINARY mode, because FB_CSVMemBufferWriter already adds CRLF! *)
                    ePath := PATH_GENERIC, tTimeout:= tTimeOut, bExecute := TRUE);
        step := 2;


    2:(* Wait until open not busy *)
        fbFileOpen( bExecute := FALSE, bError => bError, nErrID => nErrID, hFile => DestinationhFile );
        IF NOT fbFileOpen.bBusy THEN
            IF NOT fbFileOpen.bError THEN
                step := 3;
            ELSE(* Error: file not found? *)
                step := 100;
            END_IF
        END_IF

 (*   3:    (* Open Destination file *)
        fbFileOpen(  bExecute := FALSE  );
        fbFileOpen( sNetId := sNetId, sPathName := sFileName, nMode := FOPEN_MODEWRITE OR FOPEN_MODEBINARY ,(* Open file in BINARY mode, because FB_CSVMemBufferWriter already adds CRLF! *)
                        ePath := PATH_GENERIC, tTimeout:= tTimeOut, bExecute := TRUE);
        step := 4;


    4:(* Wait until open not busy *)
        fbFileOpen( bExecute := FALSE, bError => bError, nErrID => nErrID, hFile => DestinationhFile );
        IF NOT fbFileOpen.bBusy THEN
            IF NOT fbFileOpen.bError THEN
                step := 5;
            ELSE(* Error: file not found? *)
                step := 100;
            END_IF
        END_IF
*)
	(*5: 	cbReadLength:= 0;
		fbFileRead(  bExecute := FALSE  );
		fbFileRead(sNetId:= sNetId, hFile:= SourcehFile, pReadBuff:=ADR(sCSVLine), cbReadLen:= SIZEOF(sCSVLine),bExecute:= TRUE , tTimeout:= tTimeOut );
		step:= 6;
		
	6:
		fbFileRead( bExecute := FALSE, bError => bError, nErrID => nErrID, cbRead=> ReadData,bEOF=>bReadReady);
        IF NOT fbFileRead.bBusy THEN
            IF NOT fbFileRead.bError THEN
                step := 7;
            ELSE(* Error: file not found? *)
                step := 100;
            END_IF
        END_IF*)

	
    3:(* Convert one PLC record to CSV format *)
        fbWriter.eCmd := eEnumCmd_First;(* Write first field value *)
       
    FOR nRow := 1 TO 1 BY 1 DO
        str_Output:=Output[1];
                sCSVField := STRING_TO_CSVFIELD( str_Output, FALSE );(* TODO: Get field value from your application *)

					
                (* Add new field to the record buffer *)
                fbWriter(pBuffer := ADR( sCSVLine ), cbBuffer := SIZEOF( sCSVLine ), putValue := sCSVField, pValue := 0, cbValue := 0,
                            bCRLF := FALSE);(* bCRLF == TRUE => Write CRLF after the last field value *)
                IF fbWriter.bOk THEN
                    fbWriter.eCmd := eEnumCmd_Next;(* Write next field value *)
                ELSE(* Error *)
                    step := 100;
                    RETURN;
                END_IF

		  str_Output:=Output[2];
                sCSVField := STRING_TO_CSVFIELD( str_Output, FALSE );(* TODO: Get field value from your application *)


                (* Add new field to the record buffer *)
                fbWriter( pBuffer := ADR( sCSVLine ), cbBuffer := SIZEOF( sCSVLine ), putValue := sCSVField, pValue := 0, cbValue := 0,
                            bCRLF := TRUE);(* bCRLF == TRUE => Write CRLF after the last field value *)
                IF fbWriter.bOk THEN
                    fbWriter.eCmd := eEnumCmd_Next;(* Write next field value *)
                ELSE(* Error *)
                    step := 100;
                    RETURN;
                END_IF
          str_Output:=Output[5];
                sCSVField := STRING_TO_CSVFIELD( str_Output, FALSE );(* TODO: Get field value from your application *)


                (* Add new field to the record buffer *)
                fbWriter( pBuffer := ADR( sCSVLine ), cbBuffer := SIZEOF( sCSVLine ), putValue := sCSVField, pValue := 0, cbValue := 0,
                            bCRLF := FALSE);(* bCRLF == TRUE => Write CRLF after the last field value *)
                IF fbWriter.bOk THEN
                    fbWriter.eCmd := eEnumCmd_Next;(* Write next field value *)
                ELSE(* Error *)
                    step := 100;
                    RETURN;
                END_IF

		  str_Output:=Output[6];
                sCSVField := STRING_TO_CSVFIELD( str_Output, FALSE );(* TODO: Get field value from your application *)


                (* Add new field to the record buffer *)
                fbWriter(     pBuffer := ADR( sCSVLine ), cbBuffer := SIZEOF( sCSVLine ), putValue := sCSVField, pValue := 0, cbValue := 0,
                            bCRLF := TRUE);(* bCRLF == TRUE => Write CRLF after the last field value *)
                IF fbWriter.bOk THEN
                    fbWriter.eCmd := eEnumCmd_Next;(* Write next field value *)
                ELSE(* Error *)
                    step := 100;
                    RETURN;
                END_IF

  			str_Output:=Output[9];
                sCSVField := STRING_TO_CSVFIELD( str_Output, FALSE );(* TODO: Get field value from your application *)


                (* Add new field to the record buffer *)
                fbWriter(     pBuffer := ADR( sCSVLine ), cbBuffer := SIZEOF( sCSVLine ), putValue := sCSVField, pValue := 0, cbValue := 0,
                            bCRLF := FALSE);(* bCRLF == TRUE => Write CRLF after the last field value *)
                IF fbWriter.bOk THEN
                    fbWriter.eCmd := eEnumCmd_Next;(* Write next field value *)
                ELSE(* Error *)
                    step := 100;
                    RETURN;
                END_IF

		 	str_Output:=Output[10];
                sCSVField := STRING_TO_CSVFIELD( str_Output, FALSE );(* TODO: Get field value from your application *)


                (* Add new field to the record buffer *)
                fbWriter(     pBuffer := ADR( sCSVLine ), cbBuffer := SIZEOF( sCSVLine ), putValue := sCSVField, pValue := 0, cbValue := 0,
                            bCRLF := TRUE);(* bCRLF == TRUE => Write CRLF after the last field value *)
                IF fbWriter.bOk THEN
                    fbWriter.eCmd := eEnumCmd_Next;(* Write next field value *)
                ELSE(* Error *)
                    step := 100;
                    RETURN;
                END_IF
				
            str_Output:=Output[13];
                sCSVField := STRING_TO_CSVFIELD( str_Output, FALSE );(* TODO: Get field value from your application *)


                (* Add new field to the record buffer *)
                fbWriter(     pBuffer := ADR( sCSVLine ), cbBuffer := SIZEOF( sCSVLine ), putValue := sCSVField, pValue := 0, cbValue := 0,
                            bCRLF := FALSE);(* bCRLF == TRUE => Write CRLF after the last field value *)
                IF fbWriter.bOk THEN
                    fbWriter.eCmd := eEnumCmd_Next;(* Write next field value *)
                ELSE(* Error *)
                    step := 100;
                    RETURN;
                END_IF

		 	str_Output:=Output[14];
                sCSVField := STRING_TO_CSVFIELD( str_Output, FALSE );(* TODO: Get field value from your application *)


                (* Add new field to the record buffer *)
                fbWriter(     pBuffer := ADR( sCSVLine ), cbBuffer := SIZEOF( sCSVLine ), putValue := sCSVField, pValue := 0, cbValue := 0,
                            bCRLF := TRUE);(* bCRLF == TRUE => Write CRLF after the last field value *)
                IF fbWriter.bOk THEN
                    fbWriter.eCmd := eEnumCmd_Next;(* Write next field value *)
                ELSE(* Error *)
                    step := 100;
                    RETURN;
                END_IF
			
			 str_Output:=Output[17];
                sCSVField := STRING_TO_CSVFIELD( str_Output, FALSE );(* TODO: Get field value from your application *)


                (* Add new field to the record buffer *)
                fbWriter(     pBuffer := ADR( sCSVLine ), cbBuffer := SIZEOF( sCSVLine ), putValue := sCSVField, pValue := 0, cbValue := 0,
                            bCRLF := FALSE);(* bCRLF == TRUE => Write CRLF after the last field value *)
                IF fbWriter.bOk THEN
                    fbWriter.eCmd := eEnumCmd_Next;(* Write next field value *)
                ELSE(* Error *)
                    step := 100;
                    RETURN;
                END_IF

		 	str_Output:=Output[18];
                sCSVField := STRING_TO_CSVFIELD( str_Output, FALSE );(* TODO: Get field value from your application *)


                (* Add new field to the record buffer *)
                fbWriter(     pBuffer := ADR( sCSVLine ), cbBuffer := SIZEOF( sCSVLine ), putValue := sCSVField, pValue := 0, cbValue := 0,
                            bCRLF := TRUE);(* bCRLF == TRUE => Write CRLF after the last field value *)
                IF fbWriter.bOk THEN
                    fbWriter.eCmd := eEnumCmd_Next;(* Write next field value *)
                ELSE(* Error *)
                    step := 100;
                    RETURN;
                END_IF
				
			 str_Output:=Output[21];
                sCSVField := STRING_TO_CSVFIELD( str_Output, FALSE );(* TODO: Get field value from your application *)


                (* Add new field to the record buffer *)
                fbWriter(     pBuffer := ADR( sCSVLine ), cbBuffer := SIZEOF( sCSVLine ), putValue := sCSVField, pValue := 0, cbValue := 0,
                            bCRLF := FALSE);(* bCRLF == TRUE => Write CRLF after the last field value *)
                IF fbWriter.bOk THEN
                    fbWriter.eCmd := eEnumCmd_Next;(* Write next field value *)
                ELSE(* Error *)
                    step := 100;
                    RETURN;
                END_IF

		 	str_Output:=Output[22];
                sCSVField := STRING_TO_CSVFIELD( str_Output, FALSE );(* TODO: Get field value from your application *)


                (* Add new field to the record buffer *)
                fbWriter( pBuffer := ADR(sCSVLine ), cbBuffer := SIZEOF( sCSVLine ), putValue := (sCSVField), pValue := 0, cbValue := 0,
                            bCRLF := TRUE);(* bCRLF == TRUE => Write CRLF after the last field value *)
                IF fbWriter.bOk THEN
                    fbWriter.eCmd := eEnumCmd_Next;(* Write next field value *)
                ELSE(* Error *)
                    step := 100;
                    RETURN;
                END_IF
			 str_Output:=Output[25];
                sCSVField := STRING_TO_CSVFIELD( str_Output, FALSE );(* TODO: Get field value from your application *)


                (* Add new field to the record buffer *)
                fbWriter(     pBuffer := ADR( sCSVLine ), cbBuffer := SIZEOF( sCSVLine ), putValue := sCSVField, pValue := 0, cbValue := 0,
                            bCRLF := FALSE);(* bCRLF == TRUE => Write CRLF after the last field value *)
                IF fbWriter.bOk THEN
                    fbWriter.eCmd := eEnumCmd_Next;(* Write next field value *)
                ELSE(* Error *)
                    step := 100;
                    RETURN;
                END_IF

		 	str_Output:=Output[26];
                sCSVField := STRING_TO_CSVFIELD( str_Output, FALSE );(* TODO: Get field value from your application *)


                (* Add new field to the record buffer *)
                fbWriter( pBuffer := ADR(sCSVLine ), cbBuffer := SIZEOF( sCSVLine ), putValue := (sCSVField), pValue := 0, cbValue := 0,
                            bCRLF := TRUE);(* bCRLF == TRUE => Write CRLF after the last field value *)
                IF fbWriter.bOk THEN
                    fbWriter.eCmd := eEnumCmd_Next;(* Write next field value *)
                ELSE(* Error *)
                    step := 100;
                    RETURN;
                END_IF	
			str_Output:=Output[29];
                sCSVField := STRING_TO_CSVFIELD( str_Output, FALSE );(* TODO: Get field value from your application *)


                (* Add new field to the record buffer *)
                fbWriter(     pBuffer := ADR( sCSVLine ), cbBuffer := SIZEOF( sCSVLine ), putValue := sCSVField, pValue := 0, cbValue := 0,
                            bCRLF := FALSE);(* bCRLF == TRUE => Write CRLF after the last field value *)
                IF fbWriter.bOk THEN
                    fbWriter.eCmd := eEnumCmd_Next;(* Write next field value *)
                ELSE(* Error *)
                    step := 100;
                    RETURN;
                END_IF

		 	str_Output:=Output[30];
                sCSVField := STRING_TO_CSVFIELD( str_Output, FALSE );(* TODO: Get field value from your application *)


                (* Add new field to the record buffer *)
                fbWriter( pBuffer := ADR(sCSVLine ), cbBuffer := SIZEOF( sCSVLine ), putValue := (sCSVField), pValue := 0, cbValue := 0,
                            bCRLF := TRUE);(* bCRLF == TRUE => Write CRLF after the last field value *)
                IF fbWriter.bOk THEN
                    fbWriter.eCmd := eEnumCmd_Next;(* Write next field value *)
                ELSE(* Error *)
                    step := 100;
                    RETURN;
                END_IF	
			str_Output:=Output[33];
                sCSVField := STRING_TO_CSVFIELD( str_Output, FALSE );(* TODO: Get field value from your application *)


                (* Add new field to the record buffer *)
                fbWriter(     pBuffer := ADR( sCSVLine ), cbBuffer := SIZEOF( sCSVLine ), putValue := sCSVField, pValue := 0, cbValue := 0,
                            bCRLF := FALSE);(* bCRLF == TRUE => Write CRLF after the last field value *)
                IF fbWriter.bOk THEN
                    fbWriter.eCmd := eEnumCmd_Next;(* Write next field value *)
                ELSE(* Error *)
                    step := 100;
                    RETURN;
                END_IF

		 	str_Output:=Output[34];
                sCSVField := STRING_TO_CSVFIELD( str_Output, FALSE );(* TODO: Get field value from your application *)


                (* Add new field to the record buffer *)
                fbWriter( pBuffer := ADR(sCSVLine ), cbBuffer := SIZEOF( sCSVLine ), putValue := (sCSVField), pValue := 0, cbValue := 0,
                            bCRLF := TRUE);(* bCRLF == TRUE => Write CRLF after the last field value *)
                IF fbWriter.bOk THEN
                    fbWriter.eCmd := eEnumCmd_Next;(* Write next field value *)
                ELSE(* Error *)
                    step := 100;
                    RETURN;
                END_IF	
			str_Output:=Output[37];
                sCSVField := STRING_TO_CSVFIELD( str_Output, FALSE );(* TODO: Get field value from your application *)


                (* Add new field to the record buffer *)
                fbWriter(     pBuffer := ADR( sCSVLine ), cbBuffer := SIZEOF( sCSVLine ), putValue := sCSVField, pValue := 0, cbValue := 0,
                            bCRLF := FALSE);(* bCRLF == TRUE => Write CRLF after the last field value *)
                IF fbWriter.bOk THEN
                    fbWriter.eCmd := eEnumCmd_Next;(* Write next field value *)
                ELSE(* Error *)
                    step := 100;
                    RETURN;
                END_IF

		 	str_Output:=Output[38];
                sCSVField := STRING_TO_CSVFIELD( str_Output, FALSE );(* TODO: Get field value from your application *)


                (* Add new field to the record buffer *)
                fbWriter( pBuffer := ADR(sCSVLine ), cbBuffer := SIZEOF( sCSVLine ), putValue := (sCSVField), pValue := 0, cbValue := 0,
                            bCRLF := TRUE);(* bCRLF == TRUE => Write CRLF after the last field value *)
                IF fbWriter.bOk THEN
                    fbWriter.eCmd := eEnumCmd_Next;(* Write next field value *)
                ELSE(* Error *)
                    step := 100;
                    RETURN;
                END_IF	
			str_Output:=Output[41];
                sCSVField := STRING_TO_CSVFIELD( str_Output, FALSE );(* TODO: Get field value from your application *)


                (* Add new field to the record buffer *)
                fbWriter(     pBuffer := ADR( sCSVLine ), cbBuffer := SIZEOF( sCSVLine ), putValue := sCSVField, pValue := 0, cbValue := 0,
                            bCRLF := FALSE);(* bCRLF == TRUE => Write CRLF after the last field value *)
                IF fbWriter.bOk THEN
                    fbWriter.eCmd := eEnumCmd_Next;(* Write next field value *)
                ELSE(* Error *)
                    step := 100;
                    RETURN;
                END_IF

		 	str_Output:=Output[42];
                sCSVField := STRING_TO_CSVFIELD( str_Output, FALSE );(* TODO: Get field value from your application *)


                (* Add new field to the record buffer *)
                fbWriter( pBuffer := ADR(sCSVLine ), cbBuffer := SIZEOF( sCSVLine ), putValue := (sCSVField), pValue := 0, cbValue := 0,
                            bCRLF := TRUE);(* bCRLF == TRUE => Write CRLF after the last field value *)
                IF fbWriter.bOk THEN
                    fbWriter.eCmd := eEnumCmd_Next;(* Write next field value *)
                ELSE(* Error *)
                    step := 100;
                    RETURN;
                END_IF	
            END_FOR(* FOR nColumn := 0... *)

 	FOR nColumn := 1 TO 1 BY 1 DO
        str_Output:=Output[3];
                sCSVField := STRING_TO_CSVFIELD( str_Output, FALSE );(* TODO: Get field value from your application *)


                (* Add new field to the record buffer *)
                fbWriter(     pBuffer := ADR( sCSVLine ), cbBuffer := SIZEOF( sCSVLine ), putValue := sCSVField, pValue := 0, cbValue := 0,
                            bCRLF := FALSE);(* bCRLF == TRUE => Write CRLF after the last field value *)
                IF fbWriter.bOk THEN
                    fbWriter.eCmd := eEnumCmd_Next;(* Write next field value *)
                ELSE(* Error *)
                    step := 100;
                    RETURN;
                END_IF

		  str_Output:=Output[4];
                sCSVField := STRING_TO_CSVFIELD( str_Output, FALSE );(* TODO: Get field value from your application *)


                (* Add new field to the record buffer *)
                fbWriter(     pBuffer := ADR( sCSVLine ), cbBuffer := SIZEOF( sCSVLine ), putValue := sCSVField, pValue := 0, cbValue := 0,
                            bCRLF := TRUE);(* bCRLF == TRUE => Write CRLF after the last field value *)
                IF fbWriter.bOk THEN
                    fbWriter.eCmd := eEnumCmd_Next;(* Write next field value *)
                ELSE(* Error *)
                    step := 100;
                    RETURN;
                END_IF
     
		 str_Output:=Output[7];
                sCSVField := STRING_TO_CSVFIELD( str_Output, FALSE );(* TODO: Get field value from your application *)


                (* Add new field to the record buffer *)
                fbWriter(     pBuffer := ADR( sCSVLine ), cbBuffer := SIZEOF( sCSVLine ), putValue := sCSVField, pValue := 0, cbValue := 0,
                            bCRLF := FALSE);(* bCRLF == TRUE => Write CRLF after the last field value *)
                IF fbWriter.bOk THEN
                    fbWriter.eCmd := eEnumCmd_Next;(* Write next field value *)
                ELSE(* Error *)
                    step := 100;
                    RETURN;
                END_IF

		  str_Output:=Output[8];
                sCSVField := STRING_TO_CSVFIELD( str_Output, FALSE );(* TODO: Get field value from your application *)


                (* Add new field to the record buffer *)
                fbWriter(     pBuffer := ADR( sCSVLine ), cbBuffer := SIZEOF( sCSVLine ), putValue := sCSVField, pValue := 0, cbValue := 0,
                            bCRLF := TRUE);(* bCRLF == TRUE => Write CRLF after the last field value *)
                IF fbWriter.bOk THEN
                    fbWriter.eCmd := eEnumCmd_Next;(* Write next field value *)
                ELSE(* Error *)
                    step := 100;
                    RETURN;
                END_IF
			
		 str_Output:=Output[11];
                sCSVField := STRING_TO_CSVFIELD( str_Output, FALSE );(* TODO: Get field value from your application *)


                (* Add new field to the record buffer *)
                fbWriter(     pBuffer := ADR( sCSVLine ), cbBuffer := SIZEOF( sCSVLine ), putValue := sCSVField, pValue := 0, cbValue := 0,
                            bCRLF := FALSE);(* bCRLF == TRUE => Write CRLF after the last field value *)
                IF fbWriter.bOk THEN
                    fbWriter.eCmd := eEnumCmd_Next;(* Write next field value *)
                ELSE(* Error *)
                    step := 100;
                    RETURN;
                END_IF

		  str_Output:=Output[12];
                sCSVField := STRING_TO_CSVFIELD( str_Output, FALSE );(* TODO: Get field value from your application *)


                (* Add new field to the record buffer *)
                fbWriter(     pBuffer := ADR( sCSVLine ), cbBuffer := SIZEOF( sCSVLine ), putValue := sCSVField, pValue := 0, cbValue := 0,
                            bCRLF := TRUE);(* bCRLF == TRUE => Write CRLF after the last field value *)
                IF fbWriter.bOk THEN
                    fbWriter.eCmd := eEnumCmd_Next;(* Write next field value *)
                ELSE(* Error *)
                    step := 100;
                    RETURN;
                END_IF
			
			 str_Output:=Output[15];
                sCSVField := STRING_TO_CSVFIELD( str_Output, FALSE );(* TODO: Get field value from your application *)


                (* Add new field to the record buffer *)
                fbWriter(     pBuffer := ADR( sCSVLine ), cbBuffer := SIZEOF( sCSVLine ), putValue := sCSVField, pValue := 0, cbValue := 0,
                            bCRLF := FALSE);(* bCRLF == TRUE => Write CRLF after the last field value *)
                IF fbWriter.bOk THEN
                    fbWriter.eCmd := eEnumCmd_Next;(* Write next field value *)
                ELSE(* Error *)
                    step := 100;
                    RETURN;
                END_IF

		  str_Output:=Output[16];
                sCSVField := STRING_TO_CSVFIELD( str_Output, FALSE );(* TODO: Get field value from your application *)


                (* Add new field to the record buffer *)
                fbWriter(     pBuffer := ADR( sCSVLine ), cbBuffer := SIZEOF( sCSVLine ), putValue := sCSVField, pValue := 0, cbValue := 0,
                            bCRLF := TRUE);(* bCRLF == TRUE => Write CRLF after the last field value *)
                IF fbWriter.bOk THEN
                    fbWriter.eCmd := eEnumCmd_Next;(* Write next field value *)
                ELSE(* Error *)
                    step := 100;
                    RETURN;
                END_IF
			
			 str_Output:=Output[19];
                sCSVField := STRING_TO_CSVFIELD( str_Output, FALSE );(* TODO: Get field value from your application *)


                (* Add new field to the record buffer *)
                fbWriter(     pBuffer := ADR( sCSVLine ), cbBuffer := SIZEOF( sCSVLine ), putValue := sCSVField, pValue := 0, cbValue := 0,
                            bCRLF := FALSE);(* bCRLF == TRUE => Write CRLF after the last field value *)
                IF fbWriter.bOk THEN
                    fbWriter.eCmd := eEnumCmd_Next;(* Write next field value *)
                ELSE(* Error *)
                    step := 100;
                    RETURN;
                END_IF

		  str_Output:=Output[20];
                sCSVField := STRING_TO_CSVFIELD( str_Output, FALSE );(* TODO: Get field value from your application *)


                (* Add new field to the record buffer *)
                fbWriter(     pBuffer := ADR( sCSVLine ), cbBuffer := SIZEOF( sCSVLine ), putValue := sCSVField, pValue := 0, cbValue := 0,
                            bCRLF := TRUE);(* bCRLF == TRUE => Write CRLF after the last field value *)
                IF fbWriter.bOk THEN
                    fbWriter.eCmd := eEnumCmd_Next;(* Write next field value *)
                ELSE(* Error *)
                    step := 100;
                    RETURN;
                END_IF
			str_Output:=Output[23];
                sCSVField := STRING_TO_CSVFIELD( str_Output, FALSE );(* TODO: Get field value from your application *)


                (* Add new field to the record buffer *)
                fbWriter(     pBuffer := ADR( sCSVLine ), cbBuffer := SIZEOF( sCSVLine ), putValue := sCSVField, pValue := 0, cbValue := 0,
                            bCRLF := FALSE);(* bCRLF == TRUE => Write CRLF after the last field value *)
                IF fbWriter.bOk THEN
                    fbWriter.eCmd := eEnumCmd_Next;(* Write next field value *)
                ELSE(* Error *)
                    step := 100;
                    RETURN;
                END_IF

		  str_Output:=Output[24];
                sCSVField := STRING_TO_CSVFIELD( str_Output, FALSE );(* TODO: Get field value from your application *)


                (* Add new field to the record buffer *)
                fbWriter(     pBuffer := ADR( sCSVLine ), cbBuffer := SIZEOF( sCSVLine ), putValue := sCSVField, pValue := 0, cbValue := 0,
                            bCRLF := TRUE);(* bCRLF == TRUE => Write CRLF after the last field value *)
                IF fbWriter.bOk THEN
                    fbWriter.eCmd := eEnumCmd_Next;(* Write next field value *)
                ELSE(* Error *)
                    step := 100;
                    RETURN;
                END_IF
			str_Output:=Output[27];
                sCSVField := STRING_TO_CSVFIELD( str_Output, FALSE );(* TODO: Get field value from your application *)


                (* Add new field to the record buffer *)
                fbWriter(     pBuffer := ADR( sCSVLine ), cbBuffer := SIZEOF( sCSVLine ), putValue := sCSVField, pValue := 0, cbValue := 0,
                            bCRLF := FALSE);(* bCRLF == TRUE => Write CRLF after the last field value *)
                IF fbWriter.bOk THEN
                    fbWriter.eCmd := eEnumCmd_Next;(* Write next field value *)
                ELSE(* Error *)
                    step := 100;
                    RETURN;
                END_IF

		  str_Output:=Output[28];
                sCSVField := STRING_TO_CSVFIELD( str_Output, FALSE );(* TODO: Get field value from your application *)


                (* Add new field to the record buffer *)
                fbWriter(     pBuffer := ADR( sCSVLine ), cbBuffer := SIZEOF( sCSVLine ), putValue := sCSVField, pValue := 0, cbValue := 0,
                            bCRLF := TRUE);(* bCRLF == TRUE => Write CRLF after the last field value *)
                IF fbWriter.bOk THEN
                    fbWriter.eCmd := eEnumCmd_Next;(* Write next field value *)
                ELSE(* Error *)
                    step := 100;
                    RETURN;
                END_IF
			str_Output:=Output[31];
                sCSVField := STRING_TO_CSVFIELD( str_Output, FALSE );(* TODO: Get field value from your application *)


                (* Add new field to the record buffer *)
                fbWriter(     pBuffer := ADR( sCSVLine ), cbBuffer := SIZEOF( sCSVLine ), putValue := sCSVField, pValue := 0, cbValue := 0,
                            bCRLF := FALSE);(* bCRLF == TRUE => Write CRLF after the last field value *)
                IF fbWriter.bOk THEN
                    fbWriter.eCmd := eEnumCmd_Next;(* Write next field value *)
                ELSE(* Error *)
                    step := 100;
                    RETURN;
                END_IF

		  str_Output:=Output[32];
                sCSVField := STRING_TO_CSVFIELD( str_Output, FALSE );(* TODO: Get field value from your application *)


                (* Add new field to the record buffer *)
                fbWriter(     pBuffer := ADR( sCSVLine ), cbBuffer := SIZEOF( sCSVLine ), putValue := sCSVField, pValue := 0, cbValue := 0,
                            bCRLF := TRUE);(* bCRLF == TRUE => Write CRLF after the last field value *)
                IF fbWriter.bOk THEN
                    fbWriter.eCmd := eEnumCmd_Next;(* Write next field value *)
                ELSE(* Error *)
                    step := 100;
                    RETURN;
                END_IF
			str_Output:=Output[35];
                sCSVField := STRING_TO_CSVFIELD( str_Output, FALSE );(* TODO: Get field value from your application *)


                (* Add new field to the record buffer *)
                fbWriter(     pBuffer := ADR( sCSVLine ), cbBuffer := SIZEOF( sCSVLine ), putValue := sCSVField, pValue := 0, cbValue := 0,
                            bCRLF := FALSE);(* bCRLF == TRUE => Write CRLF after the last field value *)
                IF fbWriter.bOk THEN
                    fbWriter.eCmd := eEnumCmd_Next;(* Write next field value *)
                ELSE(* Error *)
                    step := 100;
                    RETURN;
                END_IF

		  str_Output:=Output[36];
                sCSVField := STRING_TO_CSVFIELD( str_Output, FALSE );(* TODO: Get field value from your application *)


                (* Add new field to the record buffer *)
                fbWriter(     pBuffer := ADR( sCSVLine ), cbBuffer := SIZEOF( sCSVLine ), putValue := sCSVField, pValue := 0, cbValue := 0,
                            bCRLF := TRUE);(* bCRLF == TRUE => Write CRLF after the last field value *)
                IF fbWriter.bOk THEN
                    fbWriter.eCmd := eEnumCmd_Next;(* Write next field value *)
                ELSE(* Error *)
                    step := 100;
                    RETURN;
                END_IF
			str_Output:=Output[39];
                sCSVField := STRING_TO_CSVFIELD( str_Output, FALSE );(* TODO: Get field value from your application *)


                (* Add new field to the record buffer *)
                fbWriter(     pBuffer := ADR( sCSVLine ), cbBuffer := SIZEOF( sCSVLine ), putValue := sCSVField, pValue := 0, cbValue := 0,
                            bCRLF := FALSE);(* bCRLF == TRUE => Write CRLF after the last field value *)
                IF fbWriter.bOk THEN
                    fbWriter.eCmd := eEnumCmd_Next;(* Write next field value *)
                ELSE(* Error *)
                    step := 100;
                    RETURN;
                END_IF

		  str_Output:=Output[40];
                sCSVField := STRING_TO_CSVFIELD( str_Output, FALSE );(* TODO: Get field value from your application *)


                (* Add new field to the record buffer *)
                fbWriter(     pBuffer := ADR( sCSVLine ), cbBuffer := SIZEOF( sCSVLine ), putValue := sCSVField, pValue := 0, cbValue := 0,
                            bCRLF := TRUE);(* bCRLF == TRUE => Write CRLF after the last field value *)
                IF fbWriter.bOk THEN
                    fbWriter.eCmd := eEnumCmd_Next;(* Write next field value *)
                ELSE(* Error *)
                    step := 100;
                    RETURN;
                END_IF
            END_FOR(* FOR nColumn := 0... *)
			fbWriter.eCmd := eEnumCmd_Next ;
            step := 10;(* Write record to the file *)
			



    10:    (* Write single text line *)
     
        fbFileWrite( bExecute := FALSE );
        fbFileWrite( sNetId := sNetId, hFile := DestinationhFile, bExecute := TRUE, pWriteBuff := ADR(sCSVLine), cbWriteLen := fbWriter.cbSize);
        step := 11;

	

    11:(* Wait until write not busy *)
        fbFileWrite( bExecute := FALSE, bError => bError, nErrID => nErrID );
        IF NOT fbFileWrite.bBusy THEN
            IF NOT fbFileWrite.bError THEN
                step := 20;(* Writing CSV-File done*)
            ELSE(* Error *)
                step := 100;
            END_IF
        END_IF


   20:    (* Close source file *)
   		
    	//IF DestinationhFile > 0  THEN
			//step:= 10;
		//ELSE
        fbFileClose( bExecute := FALSE );
        fbFileClose( sNetId := sNetId, hFile := DestinationhFile, bExecute := TRUE );
        step := 21;
		//END_IF
		



    21:(* Wait until close not busy *)
        fbFileClose( bExecute := FALSE, bError => bError, nErrID => nErrID );
			CounterPosition01.RESET:= TRUE;
			CounterPosition02.RESET:= TRUE;
			CounterPosition03.RESET:= TRUE;
			CounterPosition04.RESET:= TRUE;
			CounterPosition05.RESET:= TRUE;
			CounterPosition06.RESET:= TRUE;
			CounterPosition07.RESET:= TRUE;
			CounterPosition08.RESET:= TRUE;
			CounterPosition09.RESET:= TRUE;
			CounterPosition10.RESET:= TRUE;
        IF ( NOT fbFileClose.bBusy ) THEN
            DestinationhFile := 0;
            step := 100;
        END_IF



    100: (* Error OR ready step => cleanup *)
		
      IF ( DestinationhFile <> 0 ) THEN
           step := 20; (* Close the source file *)
        ELSE
            bBusy := FALSE;
			CounterPosition01.RESET:= FALSE;
			CounterPosition02.RESET:= FALSE;
			CounterPosition03.RESET:= FALSE;
			CounterPosition04.RESET:= FALSE;
			CounterPosition05.RESET:= FALSE;
			CounterPosition06.RESET:= FALSE;
			CounterPosition07.RESET:= FALSE;
			CounterPosition08.RESET:= FALSE;
			CounterPosition09.RESET:= FALSE;
			CounterPosition10.RESET:= FALSE;
			FileReady:= TRUE;
            step := 0;//    (* Ready *)
     END_IF




END_CASE

IF Ton1.ET = Ton1.PT AND FileReady THEN
	StartPACCounter := FALSE ;
END_IF

END_FUNCTION_BLOCK

// ---- 20_Product/20_ProBox/30_Toolbox/FB_PB_PresetEncoder.TcPOU
//Set preset value to encoder
//An ESR (Element status report telegram) is sent in order to save the status in synq database.
FUNCTION_BLOCK FB_PB_PresetEncoder
VAR_INPUT
	ElementNumber	: E_ElementNumber;					// the Functionnumber where the ESR shall be sent from
	NetId			: T_AmsNetId := ''; 				//NetId of EtherCAT Master (ex 192.31.3.1.2.1)
	SlaveAddr		: UINT := 1030; 					//Port Number of EtherCAT Slave
	Index			: WORD := 16#6003; 					//CoE Object Index
	SubIndex        : BYTE := 0; 						//Subindex of CoE Object		
	OpKeySwitch		: BOOL;							// operator key switch trigging an SDO write
	EnableWrite		: BOOL;							// endable SDO write, ie Correct conditions must be met to start writing to encoder
	PresetValue		: UDINT;
	rfbDebugMsg 	: REFERENCE TO FB_DebugMsg;		//Reference to a FB_DebugMsg object for logging purpose
END_VAR
VAR_IN_OUT
	ErrorData 		: ST_ErrorDataSet;
END_VAR


VAR_OUTPUT
END_VAR
VAR
	fbSdoWrite      : FB_EcCoESdoWrite;
	OpSwitchTmr		: TON := (PT:=T#5S);
	SdoState		: INT;	
END_VAR

VAR_TEMP
	InternalTrigger : BOOL;
	ErrType			:E_ErrorType;
	ErrParam		:STRING(system.ERROR_PARAM_STRINGLENGTH); 
	rReg			:REFERENCE TO ST_ElementRegistryConv;
END_VAR



CASE SdoState OF
	0:	//Check that op key switch is not stiched to TRUE, we need an positive edge to continue
		OpSwitchTmr(IN:=FALSE); 
		IF(OpKeySwitch=FALSE AND EnableWrite) THEN
			SdoState:=SdoState+1;
		END_IF
		
	1:	//wait for an positive edge on the operator key switch
		OpSwitchTmr(IN:=OpKeySwitch AND EnableWrite);
		IF(NOT EnableWrite) THEN
			SdoState:=0;
		ELSIF(NOT fbSdoWrite.bBusy AND OpSwitchTmr.Q) THEN
			SdoState:=SdoState+1;
		END_IF
	2: //Trigg writing
		InternalTrigger:=TRUE;
		SdoState:=SdoState+1;
	3:  //wait for writing to complete
		IF(NOT fbSdoWrite.bBusy) THEN
			SdoState:=SdoState+1;		
		END_IF
	4:  //writing complete
		IF(fbSdoWrite.bError) THEN
			ErrType := E_ErrorType.ERROR;
			ErrParam:= 'Preset Encoder FAILED';
			F_SetError(
						ErrorType 	:= E_ErrorType.ERROR, 
						ErrorParam 	:= 'Preset Encoder FAILED', 
						ErrorMsg 	:= E_ErrorConv.MAINTENANCE, 
						ErrorData 	:= ErrorData);	 
			
			fbFormatString(sFormat := 'Error while resetting encoder. Slaveaddr: %d, ADS Code: %d', arg1 := F_UINT(SlaveAddr), arg2 := F_UDINT(fbSdoWrite.nErrId));
			IF(__ISVALIDREF(rfbDebugMsg)) THEN
				rfbDebugMsg.M_SendErrorMsg(fbFormatString.sOut);
			END_IF
		ELSE
			ErrType 	:= E_ErrorType.INFO;
			ErrParam	:= 'Preset Encoder success';		
			IF(__ISVALIDREF(rfbDebugMsg)) THEN			
				rfbDebugMsg.M_SendErrorMsg('Preset encoder successfully');
			END_IF			
		END_IF
		
		
		//Send ESR 
		IF(ElementNumber > E_ElementNumber.E_BEGIN_ELEMENT AND ElementNumber < E_ElementNumber.E_END_ELEMENT) THEN
			rReg REF= ElementRegistry[ElementNumber]; 	
			
			IF( __ISVALIDREF(rReg.rElementInterface)) AND 
				__ISVALIDREF(rReg.rElementData) AND
				__ISVALIDREF(rReg.rSettingsElement) THEN
		
			//send FSR, since the ErrorType INFO or Error already being active, we need to send FSR telegram in order for it to be present in SynQ / Logging & Statistics 		
				F_ITC_SendESR(
						eChannelSrc		:= 0, 
						ElementName		:= F_ReduceToAlphaNumeric(rReg.rSettingsElement.ElementName),
						eState			:= rReg.rElementData.OperationState.eState,
						Enabled			:= rReg.rElementInterface.In.ElementEnable,
						eErrorState		:= rReg.rElementData.ErrorData.ErrorState,
						eErrorCode		:= E_ErrorConv.MAINTENANCE,
						eErrorType		:= ErrType,
						ErrorInformation:= ErrParam,
						Variable		:= 0,
						eReturnCode		:= E_ErrorConv.NO_ERROR_CODE);
			END_IF	
		END_IF
		SdoState:=SdoState+1;
		
	ELSE		
		SdoState:=0;	
END_CASE

	fbSdoWrite(
		sNetId 		:= NetId,
		nSlaveAddr 	:= SlaveAddr,
		nSubIndex	:= SubIndex, (* Subindex of CoE Object *)
		nIndex		:= Index,
		pSrcBuf     := ADR(PresetValue),
        cbBufLen    := SIZEOF(PresetValue),
		bExecute	:= InternalTrigger,
		tTimeout	:= DEFAULT_ADS_TIMEOUT);
		 
		
	OpSwitchTmr();

END_FUNCTION_BLOCK

// ---- 20_Product/20_ProBox/30_Toolbox/FB_SendTelegram.TcPOU
FUNCTION_BLOCK FB_SendTelegram  
VAR_INPUT
	FunctionNumber		: E_FunctionNumber; // FunctionNumber on which  telegram needs to be send
	ZoneNumber			: INT; 				// ZoneNumber on which zone telegram needs to be send	
END_VAR
VAR
	TransportCtrlData			:  ST_TransportControlData;	
END_VAR


TransportCtrlData := F_GetTransportControlData(FunctionNumber, ZoneNumber);

//Send IPR Telegram, internal check that zone is occupied and all addons finalized before sending telegram
METHOD PUBLIC M_SendIPR : BOOL
VAR_INPUT
	IPR_Errorcode: INT; // set Project specific error code 
	Sendtelegram: BOOL;  //Condition to send telegram
END_VAR

VAR_INST
	SendIPR  : BOOL;	// trigger when ready to send telegram
END_VAR

VAR
	ZoneData  : ST_ZoneData;
END_VAR

// Check if function number and zone is valid
IF FunctionNumber > E_FunctionNumber.F_BEGIN_FUNCTION AND
   FunctionNumber < E_FunctionNumber.F_END_FUNCTION AND
   ZoneNumber > 0 AND ZoneNumber <= NUMBER_OF_ZONES_PER_FUNCTION THEN

	/// Sent IPR
	ZoneData:= F_GetZoneData(FunctionNumber, ZoneNumber);
	IF ZoneData.AddOn.Orders.DataReady  AND
	   ZoneData.TransportControlData.Occupied  THEN 
		IF Sendtelegram AND NOT SendIPR THEN
			SendIPR:= TRUE;
			M_SendIPR:=F_ITC_SendIPR(
							eChannelSrc:= E_MFCS_Channel.AM, 
							Position:= F_ReduceToAlphaNumeric(F_GetFunctionName(FunctionNumber,ZoneNumber)), 
							TU_DataIndex:= ZoneData.TransportControlData.TU_DataIndex, 
							MSG_Sequence:= 0, 
							TU_ID:= TU_Table.TU_DataTable[ZoneData.TransportControlData.TU_DataIndex].TU_ID.ASCII, 
							TU_Type:= TU_Table.TU_DataTable[ZoneData.TransportControlData.TU_DataIndex].DataSet.TU_Type, 
							AssignmentID:= TU_Table.TU_DataTable[ZoneData.TransportControlData.TU_DataIndex].AssignmentID, 
							Height:= TU_Table.TU_DataTable[ZoneData.TransportControlData.TU_DataIndex].Profile.Height, 
							WidthRight:=  TU_Table.TU_DataTable[ZoneData.TransportControlData.TU_DataIndex].Profile.ProfileRight, 
							WidthLeft:=  TU_Table.TU_DataTable[ZoneData.TransportControlData.TU_DataIndex].Profile.ProfileLeft, 
							LengthFront:=  TU_Table.TU_DataTable[ZoneData.TransportControlData.TU_DataIndex].Profile.ProfileFront, 
							LengthRear:=  TU_Table.TU_DataTable[ZoneData.TransportControlData.TU_DataIndex].Profile.ProfileRear, 
							Weight:= TU_Table.TU_DataTable[ZoneData.TransportControlData.TU_DataIndex].Profile.Weight, 
							Tunnel:= TU_Table.TU_DataTable[ZoneData.TransportControlData.TU_DataIndex].Profile.Tunnel, 
							Runner:= TU_Table.TU_DataTable[ZoneData.TransportControlData.TU_DataIndex].Profile.Runner, 
							ErrorCode:= IPR_Errorcode, 
							ValidLabelString:= 0, 
							Label:= TU_Table.TU_DataTable[ZoneData.TransportControlData.TU_DataIndex].Label.ASCII);
		  END_IF
	END_IF
END_IF
IF NOT ZoneData.TransportControlData.Occupied THEN
	SendIPR:= FALSE;
END_IF
M_SendIPR:= SendIPR;
END_METHOD

METHOD PUBLIC M_SendMSG : BOOL
VAR_INPUT
	eMsgChannel			: E_MFCS_Channel; // Source communicaton channel	
	lMsgLength			: UDINT; // Length of structure SIZEOF/LEN
	pMsgPointer  		: PVOID; // Pointer to message structure
	Sendtelegram : BOOL; //Set to ture on the basis of condition return outside
END_VAR
VAR_INST
	SendMSG  :BOOL; // trigger when ready to send telegram
END_VAR

// Check if function number and zone is valid
IF FunctionNumber > E_FunctionNumber.F_BEGIN_FUNCTION AND
   FunctionNumber < E_FunctionNumber.F_END_FUNCTION AND
   ZoneNumber > 0 AND ZoneNumber <= NUMBER_OF_ZONES_PER_FUNCTION THEN
	/// sent MSG

	IF  Sendtelegram AND NOT SendMSG  THEN
	   SendMSG:= TRUE;
	   M_SendMSG:=F_ITC_SendMSG(eChannelSrc:= eMsgChannel, pMsgData:=pMsgPointer , Len:=lMsgLength);
	END_IF

 END_IF
M_SendMSG:=SendMSG;
END_METHOD

//Send POR0 telegram, internal check that NumberOfPresentTUs > 0 before sending telegram
METHOD PUBLIC M_SendPOR0 : BOOL
VAR_INPUT
	Sendtelegram : BOOL; //Condition to send telegram
END_VAR
VAR_INST
	SendPOR0  :BOOL; // trigger when ready to send telegram
END_VAR
VAR
	rLastTuData		: ST_LastTUdata;
END_VAR


// Check if function number and zone is valid
IF NOT(FunctionNumber > E_FunctionNumber.F_BEGIN_FUNCTION AND FunctionNumber < E_FunctionNumber.F_END_FUNCTION AND
   	   ZoneNumber > 0 AND ZoneNumber <= NUMBER_OF_ZONES_PER_FUNCTION) THEN
	   RETURN; //not valid
END_IF
//zonedata reference is valid
IF (NOT __ISVALIDREF(FunctionRegistry[FunctionNumber].Zone[ZoneNumber].refZoneData)) THEN
	RETURN; //not valid
ELSE
	rLastTuData := FunctionRegistry[FunctionNumber].Zone[ZoneNumber].refZoneData.LastTUdata;
END_IF

/// sent POR0 when TU leaving the zone
IF  TransportCtrlData.NumberOfPresentTUs =0 AND TransportCtrlData.Occupied  THEN
	IF Sendtelegram AND NOT SendPOR0 THEN
		SendPOR0 := TRUE;
		M_SendPOR0:=F_ITC_SendPOR(
					eChannelSrc:= E_MFCS_Channel.AM, 
					Position	:= F_ReduceToAlphaNumeric(F_GetFunctionName(FunctionNumber,ZoneNumber)), 
					TU_ID		:= rLastTuData.TU_ID,
					TU_Type		:= rLastTuData.TU_Type,
					AssignmentID:= rLastTuData.AssignmentID, 
					LoadInformation:=FALSE );
	END_IF
END_IF
	
//Clear flag
IF TransportCtrlData.NumberOfPresentTUs >0 OR NOT TransportCtrlData.Occupied  THEN
	SendPOR0 := FALSE;
END_IF

M_SendPOR0:= SendPOR0;
END_METHOD

//Send POR1 telegram, internal check that NumberOfPresentTUs > 0 before sending telegram
METHOD PUBLIC M_SendPOR1 : BOOL
VAR_INPUT
	Sendtelegram : BOOL; //Condition to send telegram
END_VAR

VAR_INST
	SendPOR1  :BOOL; // trigger when ready to send telegram
END_VAR

// Check if function number and zone is valid
IF FunctionNumber > E_FunctionNumber.F_BEGIN_FUNCTION AND
   FunctionNumber < E_FunctionNumber.F_END_FUNCTION AND
   ZoneNumber > 0 AND ZoneNumber <= NUMBER_OF_ZONES_PER_FUNCTION THEN

	/// sent POR1
	IF TransportCtrlData.NumberOfPresentTUs > 0  THEN
		IF Sendtelegram AND NOT SendPOR1 THEN
			SendPOR1 := TRUE;
			M_SendPOR1:=F_ITC_SendPOR(
						eChannelSrc:= E_MFCS_Channel.AM, 
						Position:=F_ReduceToAlphaNumeric(F_GetFunctionName(FunctionNumber,ZoneNumber)), 
						TU_ID:= TU_DataTable[TransportCtrlData.TU_DataIndex].TU_ID.ASCII,
						TU_Type:= TU_DataTable[TransportCtrlData.TU_DataIndex].DataSet.TU_Type,
						AssignmentID:= TU_DataTable[TransportCtrlData.TU_DataIndex].AssignmentID, 
						LoadInformation:=TRUE );
		END_IF
	END_IF
END_IF

IF TransportCtrlData.NumberOfPresentTUs = 0  THEN
	SendPOR1 := FALSE;
END_IF

M_SendPOR1:=SendPOR1;
END_METHOD

//Send TTC Telegram, internal check that zone is occupied before sending telegram
METHOD PUBLIC M_SendTTC : BOOL
VAR_INPUT
	TTC_ErroCode 		: INT :=0; 	//TTC project specific error code
	TTC_Destination		: E_FunctionNumber; // Give destination function number for exmaple if position needs to have specifc destionation to send TTC, use F_END_FUNCTION if this shall not be considered
	Sendtelegram 		: BOOL; //Condition to send telegram
END_VAR
VAR_INST
	TRIGSendTTC: BOOL; // trigger when ready to send telegram
	SendTTC :BOOL; // trigger when ready to send telegram
END_VAR
VAR
	DestinationFunction				: E_FunctionNumber;
	TU_DataIndex: INT;
END_VAR

// Check if function number and zone is valid
IF FunctionNumber > E_FunctionNumber.F_BEGIN_FUNCTION AND
   FunctionNumber < E_FunctionNumber.F_END_FUNCTION AND
   ZoneNumber > 0 AND ZoneNumber <= NUMBER_OF_ZONES_PER_FUNCTION THEN
   
	TU_DataIndex:= DINT_TO_INT(TransportCtrlData.TU_DataIndex);
	DestinationFunction := F_PB_GetTuDestination(FunctionNumber,ZoneNumber,1);
	
	IF TransportCtrlData.DataPresent AND (DestinationFunction = TTC_Destination OR TTC_Destination = E_FunctionNumber.F_END_FUNCTION) THEN
		TRIGSendTTC:= TRUE;				
	END_IF
END_IF   
 
/// send TTC
IF  TransportCtrlData.Occupied AND TRIGSendTTC  THEN
	IF  Sendtelegram AND NOT SendTTC  THEN
	   SendTTC:= TRUE;
		F_ITC_SendTTC(
					eChannelSrc				:= E_MFCS_Channel.AM,
					PositionName			:= F_ReduceToAlphaNumeric(F_GetFunctionName(FunctionNumber,ZoneNumber)),
					TU_DataIndex			:= TransportCtrlData.TU_DataIndex,
					MsgSequence				:= 0,
					TU_ID					:= TU_DataTable[TransportCtrlData.TU_DataIndex].TU_ID.ASCII,
					AssignmentID			:= TU_DataTable[TransportCtrlData.TU_DataIndex].AssignmentID,
					eReturnCode				:= TTC_ErroCode);	
	END_IF
END_IF
//clear flags if no zone data
IF NOT TransportCtrlData.Occupied THEN
	SendTTC:= FALSE;
END_IF
IF TransportCtrlData.NumberOfPresentTUs=0 THEN	
	TRIGSendTTC:= FALSE;
END_IF
M_SendTTC:=SendTTC;
END_METHOD

METHOD M_SendTTQ : BOOL
VAR_INPUT
	Sendtelegram : BOOL;	 
END_VAR
VAR_INST
	SendTTQ  :BOOL;
END_VAR

// Check if function number and zone is valid
IF FunctionNumber > E_FunctionNumber.F_BEGIN_FUNCTION AND
   FunctionNumber < E_FunctionNumber.F_END_FUNCTION AND
   ZoneNumber > 0 AND ZoneNumber <= NUMBER_OF_ZONES_PER_FUNCTION THEN
	// send TTQ
	IF(TransportCtrlData.Occupied AND TransportCtrlData.NumberOfPresentTUs>0)  THEN
		IF Sendtelegram AND NOT SendTTQ THEN
			SendTTQ := TRUE;
			M_SendTTQ:=F_ITC_SendTTQ(
						eChannelSrc		:= E_MFCS_Channel.AM, 
						PositionName	:= F_ReduceToAlphaNumeric(F_GetFunctionName(FunctionNumber,ZoneNumber)), 
						TU_DataIndex	:= TransportCtrlData.TU_DataIndex, 
						TU_ID			:= TU_DataTable[TransportCtrlData.TU_DataIndex].TU_ID.ASCII, 
						NbrOfTT			:= 1, 
						Label			:= '');
		END_IF
	ELSE
		SendTTQ := FALSE;
	END_IF
END_IF	

M_SendTTQ:= SendTTQ;
END_METHOD

END_FUNCTION_BLOCK

